LIN {X 0.007,Y -492.244,Z 296.515,A 0.000,B 0.000,C 90.000,E1 92.694} C_DIS
LIN {X -0.206,Y -481.791,Z 296.508,A 0.000,B 0.000,C 90.000,E1 91.489} C_DIS
LIN {X 0.068,Y -463.300,Z 296.496,A 0.000,B 0.000,C 90.000,E1 89.198} C_DIS
LIN {X 0.125,Y -448.239,Z 296.484,A 0.000,B 0.000,C 90.000,E1 87.135} C_DIS
LIN {X -0.046,Y -429.508,Z 296.468,A 0.000,B 0.000,C 90.000,E1 84.261} C_DIS
LIN {X 0.061,Y -414.133,Z 296.453,A 0.000,B 0.000,C 90.000,E1 81.546} C_DIS
LIN {X 0.059,Y -402.732,Z 296.441,A 0.000,B 0.000,C 90.000,E1 79.342} C_DIS
LIN {X 0.183,Y -394.078,Z 296.432,A 0.000,B 0.000,C 90.000,E1 77.645} C_DIS
LIN {X -0.138,Y -385.412,Z 296.422,A 0.000,B 0.000,C 90.000,E1 75.992} C_DIS
LIN {X -0.115,Y -373.962,Z 296.409,A 0.000,B 0.000,C 90.000,E1 73.685} C_DIS
LIN {X -0.134,Y -363.880,Z 296.398,A 0.000,B 0.000,C 90.000,E1 71.638} C_DIS
LIN {X 0.095,Y -353.920,Z 296.386,A 0.000,B 0.000,C 90.000,E1 69.518} C_DIS
LIN {X 0.073,Y -337.596,Z 296.366,A 0.000,B 0.000,C 90.000,E1 65.869} C_DIS
LIN {X 0.065,Y -324.350,Z 296.347,A 0.000,B 0.000,C 90.000,E1 62.436} C_DIS
LIN {X -0.104,Y -315.287,Z 296.333,A 0.000,B 0.000,C 90.000,E1 59.921} C_DIS
LIN {X -0.100,Y -307.615,Z 296.320,A 0.000,B 0.000,C 90.000,E1 57.661} C_DIS
LIN {X 0.046,Y -297.219,Z 296.302,A 0.000,B 0.000,C 90.000,E1 54.356} C_DIS
LIN {X 0.007,Y -289.192,Z 296.287,A 0.000,B 0.000,C 90.000,E1 51.698} C_DIS
LIN {X 0.042,Y -283.122,Z 296.276,A 0.000,B 0.000,C 90.000,E1 49.666} C_DIS
LIN {X -0.023,Y -275.077,Z 296.261,A 0.000,B 0.000,C 90.000,E1 46.944} C_DIS
LIN {X 0.007,Y -265.522,Z 296.241,A 0.000,B 0.000,C 90.000,E1 43.461} C_DIS
LIN {X -0.035,Y -259.977,Z 296.230,A 0.000,B 0.000,C 90.000,E1 41.353} C_DIS
LIN {X 0.039,Y -254.343,Z 296.218,A 0.000,B 0.000,C 90.000,E1 39.197} C_DIS
LIN {X 0.049,Y -248.620,Z 296.206,A 0.000,B 0.000,C 90.000,E1 37.030} C_DIS
LIN {X 0.150,Y -242.704,Z 296.194,A 0.000,B 0.000,C 90.000,E1 34.818} C_DIS
LIN {X 0.072,Y -234.757,Z 296.177,A 0.000,B 0.000,C 90.000,E1 31.878} C_DIS
LIN {X 0.072,Y -227.348,Z 296.160,A 0.000,B 0.000,C 90.000,E1 28.871} C_DIS
LIN {X -0.040,Y -220.568,Z 296.144,A 0.000,B 0.000,C 90.000,E1 25.848} C_DIS
LIN {X -0.103,Y -214.556,Z 296.126,A 0.000,B 0.000,C 90.000,E1 22.770} C_DIS
LIN {X -0.083,Y -209.396,Z 296.109,A 0.000,B 0.000,C 90.000,E1 19.631} C_DIS
LIN {X -0.069,Y -203.878,Z 296.087,A 0.000,B 0.000,C 90.000,E1 15.662} C_DIS
LIN {X -0.095,Y -199.386,Z 296.065,A 0.000,B 0.000,C 90.000,E1 11.658} C_DIS
LIN {X -0.019,Y -195.945,Z 296.042,A 0.000,B 0.000,C 90.000,E1 7.587} C_DIS
LIN {X -0.091,Y -192.735,Z 296.010,A 0.000,B 0.000,C 90.000,E1 1.892} C_DIS
LIN {X 0.075,Y -193.768,Z 295.924,A 0.000,B 0.000,C 90.000,E1 346.353} C_DIS
LIN {X 0.050,Y -197.101,Z 295.897,A 0.000,B 0.000,C 90.000,E1 341.456} C_DIS
LIN {X 0.012,Y -201.091,Z 295.875,A 0.000,B 0.000,C 90.000,E1 337.411} C_DIS
LIN {X 0.040,Y -206.121,Z 295.852,A 0.000,B 0.000,C 90.000,E1 333.384} C_DIS
LIN {X 0.043,Y -212.096,Z 295.830,A 0.000,B 0.000,C 90.000,E1 329.410} C_DIS
LIN {X -0.055,Y -217.536,Z 295.813,A 0.000,B 0.000,C 90.000,E1 326.294} C_DIS
LIN {X -0.005,Y -223.792,Z 295.795,A 0.000,B 0.000,C 90.000,E1 323.176} C_DIS
LIN {X -0.011,Y -230.919,Z 295.778,A 0.000,B 0.000,C 90.000,E1 320.114} C_DIS
LIN {X 0.094,Y -240.146,Z 295.760,A 0.000,B 0.000,C 90.000,E1 316.701} C_DIS
LIN {X 0.106,Y -250.567,Z 295.741,A 0.000,B 0.000,C 90.000,E1 313.380} C_DIS
LIN {X -0.081,Y -261.941,Z 295.723,A 0.000,B 0.000,C 90.000,E1 310.172} C_DIS
LIN {X -0.088,Y -274.440,Z 295.705,A 0.000,B 0.000,C 90.000,E1 306.996} C_DIS
LIN {X 0.098,Y -286.692,Z 295.690,A 0.000,B 0.000,C 90.000,E1 304.199} C_DIS
LIN {X -0.109,Y -300.388,Z 295.675,A 0.000,B 0.000,C 90.000,E1 301.544} C_DIS
LIN {X 0.043,Y -317.667,Z 295.659,A 0.000,B 0.000,C 90.000,E1 298.565} C_DIS
LIN {X -0.068,Y -338.547,Z 295.641,A 0.000,B 0.000,C 90.000,E1 295.412} C_DIS
LIN {X -0.100,Y -351.676,Z 295.631,A 0.000,B 0.000,C 90.000,E1 293.567} C_DIS
LIN {X -0.116,Y -367.035,Z 295.619,A 0.000,B 0.000,C 90.000,E1 291.461} C_DIS
LIN {X 0.211,Y -387.161,Z 295.604,A 0.000,B 0.000,C 90.000,E1 288.779} C_DIS
LIN {X 0.048,Y -400.967,Z 295.595,A 0.000,B 0.000,C 90.000,E1 287.094} C_DIS
LIN {X 0.126,Y -417.070,Z 295.584,A 0.000,B 0.000,C 90.000,E1 285.134} C_DIS
LIN {X -0.037,Y -426.115,Z 295.578,A 0.000,B 0.000,C 90.000,E1 284.064} C_DIS
LIN {X 0.045,Y -432.547,Z 295.574,A 0.000,B 0.000,C 90.000,E1 283.244} C_DIS
LIN {X -0.245,Y -438.494,Z 295.569,A 0.000,B 0.000,C 90.000,E1 282.479} C_DIS
LIN {X 0.172,Y -445.864,Z 295.563,A 0.000,B 0.000,C 90.000,E1 281.366} C_DIS
LIN {X -0.203,Y -452.680,Z 295.557,A 0.000,B 0.000,C 90.000,E1 280.366} C_DIS
LIN {X -0.143,Y -459.011,Z 295.552,A 0.000,B 0.000,C 90.000,E1 279.321} C_DIS
LIN {X -0.242,Y -466.365,Z 295.545,A 0.000,B 0.000,C 90.000,E1 278.049} C_DIS
LIN {X -0.237,Y -473.277,Z 295.537,A 0.000,B 0.000,C 90.000,E1 276.777} C_DIS
LIN {X 0.007,Y -478.221,Z 295.532,A 0.000,B 0.000,C 90.000,E1 275.739} C_DIS
LIN {X 0.151,Y -480.414,Z 295.529,A 0.000,B 0.000,C 90.000,E1 275.220} C_DIS
LIN {X -0.172,Y -482.241,Z 295.526,A 0.000,B 0.000,C 90.000,E1 274.759} C_DIS
LIN {X -0.046,Y -483.683,Z 295.524,A 0.000,B 0.000,C 90.000,E1 274.245} C_DIS
LIN {X 0.128,Y -484.744,Z 295.521,A 0.000,B 0.000,C 90.000,E1 273.726} C_DIS
LIN {X -0.207,Y -485.401,Z 295.518,A 0.000,B 0.000,C 90.000,E1 273.269} C_DIS
LIN {X -0.022,Y -485.681,Z 295.515,A 0.000,B 0.000,C 90.000,E1 272.751} C_DIS
LIN {X 0.143,Y -485.660,Z 295.513,A 0.000,B 0.000,C 90.000,E1 272.236} C_DIS
LIN {X 0.008,Y -484.956,Z 295.507,A 0.000,B 0.000,C 90.000,E1 271.260} C_DIS
LIN {X 0.174,Y -484.488,Z 295.504,A 0.000,B 0.000,C 90.000,E1 270.745} C_DIS
LIN {X -0.145,Y -483.841,Z 295.501,A 0.000,B 0.000,C 90.000,E1 270.286} C_DIS
LIN {X 0.017,Y -482.826,Z 295.499,A 0.000,B 0.000,C 90.000,E1 269.771} C_DIS
LIN {X 0.175,Y -481.325,Z 295.496,A 0.000,B 0.000,C 90.000,E1 269.255} C_DIS
LIN {X -0.155,Y -479.264,Z 295.493,A 0.000,B 0.000,C 90.000,E1 268.797} C_DIS
LIN {X -0.015,Y -476.458,Z 295.490,A 0.000,B 0.000,C 90.000,E1 268.282} C_DIS
LIN {X 0.121,Y -472.730,Z 295.488,A 0.000,B 0.000,C 90.000,E1 267.764} C_DIS
LIN {X -0.064,Y -470.502,Z 295.486,A 0.000,B 0.000,C 90.000,E1 267.535} C_DIS
LIN {X 0.094,Y -465.159,Z 295.484,A 0.000,B 0.000,C 90.000,E1 267.020} C_DIS
LIN {X -0.006,Y -462.035,Z 295.482,A 0.000,B 0.000,C 90.000,E1 266.788} C_DIS
LIN {X 0.135,Y -458.909,Z 295.481,A 0.000,B 0.000,C 90.000,E1 266.560} C_DIS
LIN {X -0.155,Y -452.026,Z 295.479,A 0.000,B 0.000,C 90.000,E1 266.216} C_DIS
LIN {X 0.191,Y -444.723,Z 295.477,A 0.000,B 0.000,C 90.000,E1 265.869} C_DIS
LIN {X 0.179,Y -436.512,Z 295.476,A 0.000,B 0.000,C 90.000,E1 265.641} C_DIS
LIN {X -0.133,Y -427.301,Z 295.475,A 0.000,B 0.000,C 90.000,E1 265.527} C_DIS
LIN {X 0.203,Y -418.825,Z 295.475,A 0.000,B 0.000,C 90.000,E1 265.412} C_DIS
LIN {X 0.062,Y -180.907,Z 295.475,A 0.000,B 0.000,C 90.000,E1 265.412} C_DIS
LIN {X -0.019,Y -180.696,Z 295.470,A 0.000,B 0.000,C 90.000,E1 264.546} C_DIS
LIN {X 0.059,Y -178.780,Z 295.442,A 0.000,B 0.000,C 90.000,E1 259.454} C_DIS
LIN {X -0.039,Y -175.826,Z 295.413,A 0.000,B 0.000,C 90.000,E1 254.393} C_DIS
LIN {X -0.038,Y -172.015,Z 295.385,A 0.000,B 0.000,C 90.000,E1 249.263} C_DIS
LIN {X -0.062,Y -171.436,Z 295.380,A 0.000,B 0.000,C 90.000,E1 248.411} C_DIS
LIN {X -0.007,Y -167.672,Z 295.356,A 0.000,B 0.000,C 90.000,E1 244.076} C_DIS
LIN {X -0.066,Y -166.346,Z 295.346,A 0.000,B 0.000,C 90.000,E1 242.359} C_DIS
LIN {X -0.074,Y -163.081,Z 295.327,A 0.000,B 0.000,C 90.000,E1 238.869} C_DIS
LIN {X -0.022,Y -161.023,Z 295.312,A 0.000,B 0.000,C 90.000,E1 236.215} C_DIS
LIN {X -0.039,Y -157.764,Z 295.293,A 0.000,B 0.000,C 90.000,E1 232.683} C_DIS
LIN {X 0.025,Y -155.802,Z 295.278,A 0.000,B 0.000,C 90.000,E1 229.989} C_DIS
LIN {X 0.079,Y -152.055,Z 295.253,A 0.000,B 0.000,C 90.000,E1 225.486} C_DIS
LIN {X -0.014,Y -150.304,Z 295.238,A 0.000,B 0.000,C 90.000,E1 222.813} C_DIS
LIN {X 0.022,Y -147.048,Z 295.213,A 0.000,B 0.000,C 90.000,E1 218.257} C_DIS
LIN {X 0.014,Y -145.627,Z 295.197,A 0.000,B 0.000,C 90.000,E1 215.518} C_DIS
LIN {X 0.012,Y -143.011,Z 295.172,A 0.000,B 0.000,C 90.000,E1 210.924} C_DIS
LIN {X -0.056,Y -141.637,Z 295.151,A 0.000,B 0.000,C 90.000,E1 207.257} C_DIS
LIN {X -0.006,Y -139.438,Z 295.115,A 0.000,B 0.000,C 90.000,E1 200.737} C_DIS
LIN {X 0.049,Y -139.170,Z 295.105,A 0.000,B 0.000,C 90.000,E1 198.852} C_DIS
LIN {X -0.055,Y -138.317,Z 295.053,A 0.000,B 0.000,C 90.000,E1 189.557} C_DIS
LIN {X -0.046,Y -139.473,Z 295.006,A 0.000,B 0.000,C 90.000,E1 181.146} C_DIS
LIN {X 0.034,Y -141.049,Z 294.975,A 0.000,B 0.000,C 90.000,E1 175.527} C_DIS
LIN {X -0.012,Y -142.420,Z 294.960,A 0.000,B 0.000,C 90.000,E1 172.761} C_DIS
LIN {X 0.050,Y -144.656,Z 294.934,A 0.000,B 0.000,C 90.000,E1 168.117} C_DIS
LIN {X -0.032,Y -147.852,Z 294.909,A 0.000,B 0.000,C 90.000,E1 163.559} C_DIS
LIN {X 0.053,Y -150.553,Z 294.888,A 0.000,B 0.000,C 90.000,E1 159.880} C_DIS
LIN {X -0.070,Y -154.020,Z 294.868,A 0.000,B 0.000,C 90.000,E1 156.305} C_DIS
LIN {X -0.011,Y -157.436,Z 294.848,A 0.000,B 0.000,C 90.000,E1 152.692} C_DIS
LIN {X 0.010,Y -161.650,Z 294.828,A 0.000,B 0.000,C 90.000,E1 149.125} C_DIS
LIN {X 0.027,Y -165.845,Z 294.809,A 0.000,B 0.000,C 90.000,E1 145.595} C_DIS
LIN {X 0.020,Y -170.819,Z 294.790,A 0.000,B 0.000,C 90.000,E1 142.110} C_DIS
LIN {X -0.064,Y -175.689,Z 294.770,A 0.000,B 0.000,C 90.000,E1 138.690} C_DIS
LIN {X 0.059,Y -181.301,Z 294.751,A 0.000,B 0.000,C 90.000,E1 135.243} C_DIS
LIN {X -0.069,Y -186.783,Z 294.733,A 0.000,B 0.000,C 90.000,E1 131.919} C_DIS
LIN {X 0.002,Y -191.375,Z 294.719,A 0.000,B 0.000,C 90.000,E1 129.402} C_DIS
LIN {X 0.085,Y -197.217,Z 294.701,A 0.000,B 0.000,C 90.000,E1 126.091} C_DIS
LIN {X 0.009,Y -200.494,Z 294.692,A 0.000,B 0.000,C 90.000,E1 124.485} C_DIS
LIN {X 0.109,Y -202.532,Z 294.685,A 0.000,B 0.000,C 90.000,E1 123.293} C_DIS
LIN {X 0.119,Y -304.407,Z 294.685,A 0.000,B 0.000,C 90.000,E1 123.293} C_DIS
LIN {X -0.015,Y -305.950,Z 294.685,A 0.000,B 0.000,C 90.000,E1 123.293} C_DIS
LIN {X -0.030,Y -310.535,Z 294.684,A 0.000,B 0.000,C 90.000,E1 123.086} C_DIS
LIN {X -0.046,Y -313.045,Z 294.683,A 0.000,B 0.000,C 90.000,E1 122.880} C_DIS
LIN {X -0.182,Y -316.856,Z 294.680,A 0.000,B 0.000,C 90.000,E1 122.418} C_DIS
LIN {X -0.123,Y -318.617,Z 294.678,A 0.000,B 0.000,C 90.000,E1 122.084} C_DIS
LIN {X 0.016,Y -321.157,Z 294.675,A 0.000,B 0.000,C 90.000,E1 121.416} C_DIS
LIN {X 0.002,Y -332.328,Z 294.659,A 0.000,B 0.000,C 90.000,E1 118.565} C_DIS
LIN {X -0.018,Y -344.918,Z 294.643,A 0.000,B 0.000,C 90.000,E1 115.771} C_DIS
LIN {X -0.013,Y -357.397,Z 294.630,A 0.000,B 0.000,C 90.000,E1 113.334} C_DIS
LIN {X 0.185,Y -371.181,Z 294.616,A 0.000,B 0.000,C 90.000,E1 110.918} C_DIS
LIN {X 0.115,Y -386.373,Z 294.603,A 0.000,B 0.000,C 90.000,E1 108.598} C_DIS
LIN {X 0.171,Y -403.084,Z 294.591,A 0.000,B 0.000,C 90.000,E1 106.315} C_DIS
LIN {X 0.025,Y -421.438,Z 294.578,A 0.000,B 0.000,C 90.000,E1 104.120} C_DIS
LIN {X -0.070,Y -441.277,Z 294.567,A 0.000,B 0.000,C 90.000,E1 102.007} C_DIS
LIN {X 0.214,Y -461.762,Z 294.556,A 0.000,B 0.000,C 90.000,E1 100.018} C_DIS
LIN {X -0.085,Y -485.422,Z 294.545,A 0.000,B 0.000,C 90.000,E1 98.049} C_DIS
LIN {X 0.021,Y -498.737,Z 294.539,A 0.000,B 0.000,C 90.000,E1 97.004} C_DIS
LIN {X 0.249,Y -500.822,Z 294.538,A 0.000,B 0.000,C 90.000,E1 96.777} C_DIS
LIN {X 0.176,Y -502.677,Z 294.536,A 0.000,B 0.000,C 90.000,E1 96.549} C_DIS
LIN {X 0.158,Y -504.077,Z 294.535,A 0.000,B 0.000,C 90.000,E1 96.315} C_DIS
LIN {X -0.042,Y -505.916,Z 294.533,A 0.000,B 0.000,C 90.000,E1 95.853} C_DIS
LIN {X 0.269,Y -506.626,Z 294.530,A 0.000,B 0.000,C 90.000,E1 95.334} C_DIS
LIN {X 0.040,Y -506.327,Z 294.527,A 0.000,B 0.000,C 90.000,E1 94.878} C_DIS
LIN {X -0.139,Y -504.971,Z 294.524,A 0.000,B 0.000,C 90.000,E1 94.416} C_DIS
LIN {X -0.249,Y -503.823,Z 294.523,A 0.000,B 0.000,C 90.000,E1 94.188} C_DIS
LIN {X 0.178,Y -502.279,Z 294.522,A 0.000,B 0.000,C 90.000,E1 93.898} C_DIS
LIN {X 0.226,Y -494.728,Z 294.516,A 0.000,B 0.000,C 90.000,E1 92.922} C_DIS
LIN {X 0.036,Y -484.399,Z 294.510,A 0.000,B 0.000,C 90.000,E1 91.718} C_DIS
LIN {X 0.167,Y -463.746,Z 294.496,A 0.000,B 0.000,C 90.000,E1 89.198} C_DIS
LIN {X -0.216,Y -448.648,Z 294.484,A 0.000,B 0.000,C 90.000,E1 87.192} C_DIS
LIN {X -0.227,Y -428.267,Z 294.467,A 0.000,B 0.000,C 90.000,E1 84.033} C_DIS
LIN {X -0.095,Y -413.022,Z 294.452,A 0.000,B 0.000,C 90.000,E1 81.310} C_DIS
LIN {X -0.114,Y -401.654,Z 294.439,A 0.000,B 0.000,C 90.000,E1 79.106} C_DIS
LIN {X 0.063,Y -391.543,Z 294.428,A 0.000,B 0.000,C 90.000,E1 77.117} C_DIS
LIN {X -0.139,Y -380.032,Z 294.416,A 0.000,B 0.000,C 90.000,E1 74.866} C_DIS
LIN {X -0.132,Y -370.007,Z 294.405,A 0.000,B 0.000,C 90.000,E1 72.834} C_DIS
LIN {X 0.184,Y -358.557,Z 294.391,A 0.000,B 0.000,C 90.000,E1 70.423} C_DIS
LIN {X 0.017,Y -345.956,Z 294.376,A 0.000,B 0.000,C 90.000,E1 67.741} C_DIS
LIN {X 0.035,Y -334.235,Z 294.361,A 0.000,B 0.000,C 90.000,E1 64.973} C_DIS
LIN {X 0.078,Y -321.330,Z 294.342,A 0.000,B 0.000,C 90.000,E1 61.513} C_DIS
LIN {X -0.037,Y -310.212,Z 294.324,A 0.000,B 0.000,C 90.000,E1 58.329} C_DIS
LIN {X 0.030,Y -299.658,Z 294.306,A 0.000,B 0.000,C 90.000,E1 55.055} C_DIS
LIN {X 0.054,Y -291.573,Z 294.291,A 0.000,B 0.000,C 90.000,E1 52.396} C_DIS
LIN {X 0.177,Y -285.517,Z 294.280,A 0.000,B 0.000,C 90.000,E1 50.356} C_DIS
LIN {X -0.039,Y -277.399,Z 294.265,A 0.000,B 0.000,C 90.000,E1 47.676} C_DIS
LIN {X 0.075,Y -267.698,Z 294.246,A 0.000,B 0.000,C 90.000,E1 44.190} C_DIS
LIN {X 0.077,Y -262.142,Z 294.234,A 0.000,B 0.000,C 90.000,E1 42.081} C_DIS
LIN {X -0.001,Y -256.552,Z 294.222,A 0.000,B 0.000,C 90.000,E1 39.967} C_DIS
LIN {X 0.013,Y -250.884,Z 294.210,A 0.000,B 0.000,C 90.000,E1 37.810} C_DIS
LIN {X -0.043,Y -245.007,Z 294.198,A 0.000,B 0.000,C 90.000,E1 35.644} C_DIS
LIN {X 0.043,Y -239.047,Z 294.186,A 0.000,B 0.000,C 90.000,E1 33.420} C_DIS
LIN {X -0.050,Y -231.258,Z 294.169,A 0.000,B 0.000,C 90.000,E1 30.463} C_DIS
LIN {X -0.035,Y -222.505,Z 294.148,A 0.000,B 0.000,C 90.000,E1 26.668} C_DIS
LIN {X -0.088,Y -214.899,Z 294.127,A 0.000,B 0.000,C 90.000,E1 22.823} C_DIS
LIN {X -0.063,Y -209.719,Z 294.109,A 0.000,B 0.000,C 90.000,E1 19.685} C_DIS
LIN {X -0.045,Y -204.183,Z 294.087,A 0.000,B 0.000,C 90.000,E1 15.717} C_DIS
LIN {X -0.065,Y -199.679,Z 294.065,A 0.000,B 0.000,C 90.000,E1 11.715} C_DIS
LIN {X 0.017,Y -196.219,Z 294.042,A 0.000,B 0.000,C 90.000,E1 7.644} C_DIS
LIN {X -0.046,Y -192.989,Z 294.011,A 0.000,B 0.000,C 90.000,E1 1.949} C_DIS
LIN {X -0.093,Y -193.946,Z 293.924,A 0.000,B 0.000,C 90.000,E1 346.408} C_DIS
LIN {X 0.076,Y -197.236,Z 293.897,A 0.000,B 0.000,C 90.000,E1 341.456} C_DIS
LIN {X 0.043,Y -201.224,Z 293.875,A 0.000,B 0.000,C 90.000,E1 337.411} C_DIS
LIN {X 0.077,Y -206.253,Z 293.852,A 0.000,B 0.000,C 90.000,E1 333.384} C_DIS
LIN {X 0.085,Y -212.202,Z 293.830,A 0.000,B 0.000,C 90.000,E1 329.410} C_DIS
LIN {X -0.010,Y -217.665,Z 293.813,A 0.000,B 0.000,C 90.000,E1 326.294} C_DIS
LIN {X -0.089,Y -223.938,Z 293.795,A 0.000,B 0.000,C 90.000,E1 323.210} C_DIS
LIN {X 0.045,Y -231.110,Z 293.778,A 0.000,B 0.000,C 90.000,E1 320.114} C_DIS
LIN {X -0.017,Y -240.364,Z 293.760,A 0.000,B 0.000,C 90.000,E1 316.743} C_DIS
LIN {X 0.007,Y -250.757,Z 293.741,A 0.000,B 0.000,C 90.000,E1 313.419} C_DIS
LIN {X 0.000,Y -262.119,Z 293.723,A 0.000,B 0.000,C 90.000,E1 310.172} C_DIS
LIN {X 0.003,Y -274.632,Z 293.706,A 0.000,B 0.000,C 90.000,E1 306.996} C_DIS
LIN {X -0.039,Y -286.899,Z 293.690,A 0.000,B 0.000,C 90.000,E1 304.246} C_DIS
LIN {X 0.000,Y -300.617,Z 293.675,A 0.000,B 0.000,C 90.000,E1 301.544} C_DIS
LIN {X -0.113,Y -317.889,Z 293.659,A 0.000,B 0.000,C 90.000,E1 298.615} C_DIS
LIN {X 0.070,Y -338.772,Z 293.641,A 0.000,B 0.000,C 90.000,E1 295.412} C_DIS
LIN {X 0.047,Y -351.870,Z 293.631,A 0.000,B 0.000,C 90.000,E1 293.567} C_DIS
LIN {X 0.042,Y -367.202,Z 293.619,A 0.000,B 0.000,C 90.000,E1 291.461} C_DIS
LIN {X 0.027,Y -389.558,Z 293.603,A 0.000,B 0.000,C 90.000,E1 288.544} C_DIS
LIN {X -0.096,Y -403.296,Z 293.594,A 0.000,B 0.000,C 90.000,E1 286.858} C_DIS
LIN {X 0.036,Y -419.280,Z 293.583,A 0.000,B 0.000,C 90.000,E1 284.898} C_DIS
LIN {X -0.102,Y -428.214,Z 293.577,A 0.000,B 0.000,C 90.000,E1 283.828} C_DIS
LIN {X -0.009,Y -434.477,Z 293.572,A 0.000,B 0.000,C 90.000,E1 283.008} C_DIS
LIN {X -0.072,Y -442.119,Z 293.566,A 0.000,B 0.000,C 90.000,E1 281.951} C_DIS
LIN {X -0.048,Y -449.158,Z 293.560,A 0.000,B 0.000,C 90.000,E1 280.894} C_DIS
LIN {X -0.026,Y -455.719,Z 293.555,A 0.000,B 0.000,C 90.000,E1 279.849} C_DIS
LIN {X -0.097,Y -463.283,Z 293.548,A 0.000,B 0.000,C 90.000,E1 278.568} C_DIS
LIN {X 0.116,Y -471.739,Z 293.539,A 0.000,B 0.000,C 90.000,E1 277.011} C_DIS
LIN {X -0.125,Y -476.861,Z 293.533,A 0.000,B 0.000,C 90.000,E1 276.030} C_DIS
LIN {X -0.130,Y -480.211,Z 293.529,A 0.000,B 0.000,C 90.000,E1 275.277} C_DIS
LIN {X 0.024,Y -482.082,Z 293.526,A 0.000,B 0.000,C 90.000,E1 274.759} C_DIS
LIN {X 0.148,Y -483.513,Z 293.524,A 0.000,B 0.000,C 90.000,E1 274.245} C_DIS
LIN {X -0.162,Y -484.596,Z 293.521,A 0.000,B 0.000,C 90.000,E1 273.784} C_DIS
LIN {X -0.012,Y -485.230,Z 293.518,A 0.000,B 0.000,C 90.000,E1 273.269} C_DIS
LIN {X 0.171,Y -485.559,Z 293.515,A 0.000,B 0.000,C 90.000,E1 272.751} C_DIS
LIN {X -0.151,Y -485.544,Z 293.513,A 0.000,B 0.000,C 90.000,E1 272.293} C_DIS
LIN {X 0.198,Y -484.896,Z 293.507,A 0.000,B 0.000,C 90.000,E1 271.260} C_DIS
LIN {X 0.044,Y -483.782,Z 293.502,A 0.000,B 0.000,C 90.000,E1 270.286} C_DIS
LIN {X 0.205,Y -482.822,Z 293.499,A 0.000,B 0.000,C 90.000,E1 269.771} C_DIS
LIN {X -0.119,Y -481.361,Z 293.496,A 0.000,B 0.000,C 90.000,E1 269.312} C_DIS
LIN {X 0.032,Y -479.303,Z 293.493,A 0.000,B 0.000,C 90.000,E1 268.797} C_DIS
LIN {X 0.172,Y -476.535,Z 293.491,A 0.000,B 0.000,C 90.000,E1 268.282} C_DIS
LIN {X 0.009,Y -474.850,Z 293.489,A 0.000,B 0.000,C 90.000,E1 268.051} C_DIS
LIN {X 0.121,Y -470.648,Z 293.486,A 0.000,B 0.000,C 90.000,E1 267.535} C_DIS
LIN {X -0.065,Y -468.184,Z 293.485,A 0.000,B 0.000,C 90.000,E1 267.306} C_DIS
LIN {X -0.240,Y -465.387,Z 293.484,A 0.000,B 0.000,C 90.000,E1 267.078} C_DIS
LIN {X 0.073,Y -462.253,Z 293.482,A 0.000,B 0.000,C 90.000,E1 266.788} C_DIS
LIN {X 0.186,Y -459.176,Z 293.481,A 0.000,B 0.000,C 90.000,E1 266.560} C_DIS
LIN {X -0.157,Y -455.611,Z 293.480,A 0.000,B 0.000,C 90.000,E1 266.388} C_DIS
LIN {X -0.188,Y -448.440,Z 293.478,A 0.000,B 0.000,C 90.000,E1 266.045} C_DIS
LIN {X 0.114,Y -444.902,Z 293.477,A 0.000,B 0.000,C 90.000,E1 265.869} C_DIS
LIN {X 0.077,Y -436.623,Z 293.476,A 0.000,B 0.000,C 90.000,E1 265.641} C_DIS
LIN {X 0.181,Y -427.335,Z 293.475,A 0.000,B 0.000,C 90.000,E1 265.469} C_DIS
LIN {X 0.083,Y -417.648,Z 293.475,A 0.000,B 0.000,C 90.000,E1 265.412} C_DIS
LIN {X 0.008,Y -180.906,Z 293.475,A 0.000,B 0.000,C 90.000,E1 265.412} C_DIS
LIN {X 0.089,Y -180.684,Z 293.470,A 0.000,B 0.000,C 90.000,E1 264.489} C_DIS
LIN {X -0.013,Y -178.767,Z 293.441,A 0.000,B 0.000,C 90.000,E1 259.454} C_DIS
LIN {X 0.059,Y -175.814,Z 293.413,A 0.000,B 0.000,C 90.000,E1 254.338} C_DIS
LIN {X 0.052,Y -172.001,Z 293.385,A 0.000,B 0.000,C 90.000,E1 249.209} C_DIS
LIN {X 0.027,Y -171.416,Z 293.380,A 0.000,B 0.000,C 90.000,E1 248.358} C_DIS
LIN {X 0.074,Y -167.654,Z 293.356,A 0.000,B 0.000,C 90.000,E1 244.024} C_DIS
LIN {X 0.089,Y -166.321,Z 293.346,A 0.000,B 0.000,C 90.000,E1 242.281} C_DIS
LIN {X -0.002,Y -163.061,Z 293.327,A 0.000,B 0.000,C 90.000,E1 238.820} C_DIS
LIN {X 0.043,Y -160.998,Z 293.312,A 0.000,B 0.000,C 90.000,E1 236.167} C_DIS
LIN {X 0.020,Y -157.744,Z 293.292,A 0.000,B 0.000,C 90.000,E1 232.637} C_DIS
LIN {X -0.041,Y -155.783,Z 293.278,A 0.000,B 0.000,C 90.000,E1 229.989} C_DIS
LIN {X 0.014,Y -152.036,Z 293.253,A 0.000,B 0.000,C 90.000,E1 225.486} C_DIS
LIN {X 0.032,Y -150.285,Z 293.238,A 0.000,B 0.000,C 90.000,E1 222.771} C_DIS
LIN {X -0.043,Y -147.035,Z 293.212,A 0.000,B 0.000,C 90.000,E1 218.257} C_DIS
LIN {X -0.050,Y -145.615,Z 293.197,A 0.000,B 0.000,C 90.000,E1 215.518} C_DIS
LIN {X -0.050,Y -142.999,Z 293.172,A 0.000,B 0.000,C 90.000,E1 210.924} C_DIS
LIN {X 0.007,Y -141.626,Z 293.151,A 0.000,B 0.000,C 90.000,E1 207.206} C_DIS
LIN {X -0.068,Y -139.433,Z 293.115,A 0.000,B 0.000,C 90.000,E1 200.737} C_DIS
LIN {X -0.014,Y -139.165,Z 293.105,A 0.000,B 0.000,C 90.000,E1 198.852} C_DIS
LIN {X 0.019,Y -138.316,Z 293.053,A 0.000,B 0.000,C 90.000,E1 189.500} C_DIS
LIN {X 0.031,Y -139.477,Z 293.006,A 0.000,B 0.000,C 90.000,E1 181.088} C_DIS
LIN {X -0.028,Y -141.060,Z 292.975,A 0.000,B 0.000,C 90.000,E1 175.527} C_DIS
LIN {X 0.067,Y -142.433,Z 292.960,A 0.000,B 0.000,C 90.000,E1 172.704} C_DIS
LIN {X -0.013,Y -144.671,Z 292.934,A 0.000,B 0.000,C 90.000,E1 168.117} C_DIS
LIN {X -0.030,Y -147.256,Z 292.914,A 0.000,B 0.000,C 90.000,E1 164.448} C_DIS
LIN {X -0.013,Y -150.574,Z 292.888,A 0.000,B 0.000,C 90.000,E1 159.880} C_DIS
LIN {X 0.066,Y -154.044,Z 292.868,A 0.000,B 0.000,C 90.000,E1 156.230} C_DIS
LIN {X -0.007,Y -157.462,Z 292.848,A 0.000,B 0.000,C 90.000,E1 152.666} C_DIS
LIN {X -0.059,Y -161.682,Z 292.828,A 0.000,B 0.000,C 90.000,E1 149.125} C_DIS
LIN {X -0.042,Y -165.877,Z 292.809,A 0.000,B 0.000,C 90.000,E1 145.595} C_DIS
LIN {X -0.051,Y -170.855,Z 292.789,A 0.000,B 0.000,C 90.000,E1 142.110} C_DIS
LIN {X -0.004,Y -175.725,Z 292.770,A 0.000,B 0.000,C 90.000,E1 138.647} C_DIS
LIN {X -0.014,Y -181.336,Z 292.751,A 0.000,B 0.000,C 90.000,E1 135.243} C_DIS
LIN {X -0.019,Y -186.823,Z 292.733,A 0.000,B 0.000,C 90.000,E1 131.881} C_DIS
LIN {X 0.075,Y -191.412,Z 292.719,A 0.000,B 0.000,C 90.000,E1 129.358} C_DIS
LIN {X 0.008,Y -197.260,Z 292.701,A 0.000,B 0.000,C 90.000,E1 126.091} C_DIS
LIN {X -0.068,Y -200.538,Z 292.691,A 0.000,B 0.000,C 90.000,E1 124.485} C_DIS
LIN {X -0.030,Y -202.602,Z 292.685,A 0.000,B 0.000,C 90.000,E1 123.293} C_DIS
LIN {X -0.089,Y -304.500,Z 292.685,A 0.000,B 0.000,C 90.000,E1 123.293} C_DIS
LIN {X 0.110,Y -310.380,Z 292.684,A 0.000,B 0.000,C 90.000,E1 123.038} C_DIS
LIN {X 0.096,Y -312.969,Z 292.682,A 0.000,B 0.000,C 90.000,E1 122.832} C_DIS
LIN {X 0.202,Y -316.775,Z 292.680,A 0.000,B 0.000,C 90.000,E1 122.339} C_DIS
LIN {X -0.008,Y -318.585,Z 292.678,A 0.000,B 0.000,C 90.000,E1 122.054} C_DIS
LIN {X -0.038,Y -321.171,Z 292.674,A 0.000,B 0.000,C 90.000,E1 121.416} C_DIS
LIN {X -0.053,Y -332.347,Z 292.659,A 0.000,B 0.000,C 90.000,E1 118.565} C_DIS
LIN {X -0.076,Y -344.941,Z 292.643,A 0.000,B 0.000,C 90.000,E1 115.771} C_DIS
LIN {X -0.072,Y -357.425,Z 292.630,A 0.000,B 0.000,C 90.000,E1 113.334} C_DIS
LIN {X 0.124,Y -371.214,Z 292.616,A 0.000,B 0.000,C 90.000,E1 110.918} C_DIS
LIN {X 0.052,Y -386.411,Z 292.603,A 0.000,B 0.000,C 90.000,E1 108.598} C_DIS
LIN {X 0.107,Y -403.128,Z 292.591,A 0.000,B 0.000,C 90.000,E1 106.315} C_DIS
LIN {X -0.041,Y -421.490,Z 292.578,A 0.000,B 0.000,C 90.000,E1 104.120} C_DIS
LIN {X -0.135,Y -441.333,Z 292.567,A 0.000,B 0.000,C 90.000,E1 102.007} C_DIS
LIN {X 0.151,Y -461.819,Z 292.556,A 0.000,B 0.000,C 90.000,E1 100.018} C_DIS
LIN {X -0.147,Y -485.482,Z 292.545,A 0.000,B 0.000,C 90.000,E1 98.049} C_DIS
LIN {X -0.041,Y -498.817,Z 292.539,A 0.000,B 0.000,C 90.000,E1 97.004} C_DIS
LIN {X 0.188,Y -500.942,Z 292.538,A 0.000,B 0.000,C 90.000,E1 96.777} C_DIS
LIN {X 0.138,Y -502.807,Z 292.536,A 0.000,B 0.000,C 90.000,E1 96.549} C_DIS
LIN {X 0.144,Y -504.220,Z 292.535,A 0.000,B 0.000,C 90.000,E1 96.315} C_DIS
LIN {X -0.055,Y -506.099,Z 292.532,A 0.000,B 0.000,C 90.000,E1 95.853} C_DIS
LIN {X 0.256,Y -506.844,Z 292.530,A 0.000,B 0.000,C 90.000,E1 95.334} C_DIS
LIN {X 0.028,Y -506.581,Z 292.527,A 0.000,B 0.000,C 90.000,E1 94.878} C_DIS
LIN {X -0.150,Y -505.265,Z 292.524,A 0.000,B 0.000,C 90.000,E1 94.416} C_DIS
LIN {X -0.259,Y -504.142,Z 292.523,A 0.000,B 0.000,C 90.000,E1 94.188} C_DIS
LIN {X 0.169,Y -502.628,Z 292.522,A 0.000,B 0.000,C 90.000,E1 93.898} C_DIS
LIN {X -0.180,Y -497.073,Z 292.518,A 0.000,B 0.000,C 90.000,E1 93.212} C_DIS
LIN {X -0.180,Y -489.032,Z 292.512,A 0.000,B 0.000,C 90.000,E1 92.236} C_DIS
LIN {X -0.086,Y -466.089,Z 292.497,A 0.000,B 0.000,C 90.000,E1 89.484} C_DIS
LIN {X -0.181,Y -452.605,Z 292.487,A 0.000,B 0.000,C 90.000,E1 87.707} C_DIS
LIN {X 0.197,Y -433.472,Z 292.471,A 0.000,B 0.000,C 90.000,E1 84.780} C_DIS
LIN {X -0.063,Y -417.699,Z 292.456,A 0.000,B 0.000,C 90.000,E1 82.129} C_DIS
LIN {X 0.120,Y -404.773,Z 292.443,A 0.000,B 0.000,C 90.000,E1 79.634} C_DIS
LIN {X -0.109,Y -396.170,Z 292.433,A 0.000,B 0.000,C 90.000,E1 77.993} C_DIS
LIN {X 0.043,Y -386.081,Z 292.422,A 0.000,B 0.000,C 90.000,E1 75.992} C_DIS
LIN {X 0.077,Y -374.626,Z 292.409,A 0.000,B 0.000,C 90.000,E1 73.685} C_DIS
LIN {X 0.067,Y -364.566,Z 292.398,A 0.000,B 0.000,C 90.000,E1 71.638} C_DIS
LIN {X 0.022,Y -353.232,Z 292.385,A 0.000,B 0.000,C 90.000,E1 69.263} C_DIS
LIN {X -0.012,Y -337.089,Z 292.365,A 0.000,B 0.000,C 90.000,E1 65.613} C_DIS
LIN {X 0.123,Y -323.953,Z 292.345,A 0.000,B 0.000,C 90.000,E1 62.153} C_DIS
LIN {X 0.067,Y -314.936,Z 292.331,A 0.000,B 0.000,C 90.000,E1 59.616} C_DIS
LIN {X 0.010,Y -306.224,Z 292.317,A 0.000,B 0.000,C 90.000,E1 57.041} C_DIS
LIN {X 0.095,Y -297.963,Z 292.302,A 0.000,B 0.000,C 90.000,E1 54.402} C_DIS
LIN {X -0.017,Y -291.910,Z 292.291,A 0.000,B 0.000,C 90.000,E1 52.431} C_DIS
LIN {X -0.115,Y -285.834,Z 292.280,A 0.000,B 0.000,C 90.000,E1 50.436} C_DIS
LIN {X -0.111,Y -277.690,Z 292.265,A 0.000,B 0.000,C 90.000,E1 47.715} C_DIS
LIN {X 0.003,Y -267.964,Z 292.246,A 0.000,B 0.000,C 90.000,E1 44.231} C_DIS
LIN {X -0.077,Y -260.560,Z 292.230,A 0.000,B 0.000,C 90.000,E1 41.434} C_DIS
LIN {X 0.009,Y -254.941,Z 292.218,A 0.000,B 0.000,C 90.000,E1 39.277} C_DIS
LIN {X 0.035,Y -249.256,Z 292.206,A 0.000,B 0.000,C 90.000,E1 37.111} C_DIS
LIN {X -0.051,Y -243.321,Z 292.194,A 0.000,B 0.000,C 90.000,E1 34.945} C_DIS
LIN {X -0.110,Y -235.368,Z 292.178,A 0.000,B 0.000,C 90.000,E1 32.005} C_DIS
LIN {X 0.108,Y -227.950,Z 292.161,A 0.000,B 0.000,C 90.000,E1 28.949} C_DIS
LIN {X 0.015,Y -221.205,Z 292.144,A 0.000,B 0.000,C 90.000,E1 25.924} C_DIS
LIN {X 0.055,Y -215.207,Z 292.127,A 0.000,B 0.000,C 90.000,E1 22.823} C_DIS
LIN {X 0.013,Y -210.013,Z 292.109,A 0.000,B 0.000,C 90.000,E1 19.704} C_DIS
LIN {X 0.051,Y -204.461,Z 292.087,A 0.000,B 0.000,C 90.000,E1 15.733} C_DIS
LIN {X 0.091,Y -199.945,Z 292.065,A 0.000,B 0.000,C 90.000,E1 11.715} C_DIS
LIN {X -0.025,Y -195.882,Z 292.038,A 0.000,B 0.000,C 90.000,E1 6.891} C_DIS
LIN {X 0.070,Y -192.920,Z 292.006,A 0.000,B 0.000,C 90.000,E1 1.146} C_DIS
LIN {X -0.074,Y -194.121,Z 291.924,A 0.000,B 0.000,C 90.000,E1 346.408} C_DIS
LIN {X 0.103,Y -197.383,Z 291.897,A 0.000,B 0.000,C 90.000,E1 341.456} C_DIS
LIN {X 0.075,Y -201.360,Z 291.875,A 0.000,B 0.000,C 90.000,E1 337.411} C_DIS
LIN {X 0.114,Y -206.386,Z 291.852,A 0.000,B 0.000,C 90.000,E1 333.384} C_DIS
LIN {X -0.056,Y -212.320,Z 291.830,A 0.000,B 0.000,C 90.000,E1 329.459} C_DIS
LIN {X 0.036,Y -217.796,Z 291.813,A 0.000,B 0.000,C 90.000,E1 326.294} C_DIS
LIN {X -0.038,Y -224.089,Z 291.796,A 0.000,B 0.000,C 90.000,E1 323.210} C_DIS
LIN {X -0.047,Y -231.302,Z 291.779,A 0.000,B 0.000,C 90.000,E1 320.150} C_DIS
LIN {X 0.047,Y -240.580,Z 291.760,A 0.000,B 0.000,C 90.000,E1 316.743} C_DIS
LIN {X -0.102,Y -250.951,Z 291.741,A 0.000,B 0.000,C 90.000,E1 313.461} C_DIS
LIN {X 0.083,Y -262.304,Z 291.723,A 0.000,B 0.000,C 90.000,E1 310.172} C_DIS
LIN {X -0.071,Y -274.816,Z 291.706,A 0.000,B 0.000,C 90.000,E1 307.030} C_DIS
LIN {X 0.061,Y -287.103,Z 291.690,A 0.000,B 0.000,C 90.000,E1 304.246} C_DIS
LIN {X 0.107,Y -299.024,Z 291.677,A 0.000,B 0.000,C 90.000,E1 301.878} C_DIS
LIN {X 0.011,Y -318.113,Z 291.659,A 0.000,B 0.000,C 90.000,E1 298.615} C_DIS
LIN {X -0.075,Y -336.840,Z 291.643,A 0.000,B 0.000,C 90.000,E1 295.771} C_DIS
LIN {X 0.056,Y -352.032,Z 291.631,A 0.000,B 0.000,C 90.000,E1 293.590} C_DIS
LIN {X 0.067,Y -367.354,Z 291.619,A 0.000,B 0.000,C 90.000,E1 291.482} C_DIS
LIN {X 0.062,Y -387.323,Z 291.605,A 0.000,B 0.000,C 90.000,E1 288.852} C_DIS
LIN {X 0.021,Y -401.056,Z 291.595,A 0.000,B 0.000,C 90.000,E1 287.149} C_DIS
LIN {X 0.096,Y -416.951,Z 291.584,A 0.000,B 0.000,C 90.000,E1 285.190} C_DIS
LIN {X 0.089,Y -428.112,Z 291.577,A 0.000,B 0.000,C 90.000,E1 283.828} C_DIS
LIN {X 0.184,Y -434.367,Z 291.572,A 0.000,B 0.000,C 90.000,E1 283.008} C_DIS
LIN {X 0.123,Y -441.967,Z 291.566,A 0.000,B 0.000,C 90.000,E1 281.951} C_DIS
LIN {X 0.148,Y -448.969,Z 291.561,A 0.000,B 0.000,C 90.000,E1 280.894} C_DIS
LIN {X 0.170,Y -455.524,Z 291.555,A 0.000,B 0.000,C 90.000,E1 279.849} C_DIS
LIN {X 0.100,Y -463.066,Z 291.548,A 0.000,B 0.000,C 90.000,E1 278.568} C_DIS
LIN {X 0.060,Y -470.156,Z 291.541,A 0.000,B 0.000,C 90.000,E1 277.296} C_DIS
LIN {X -0.202,Y -475.407,Z 291.535,A 0.000,B 0.000,C 90.000,E1 276.315} C_DIS
LIN {X 0.066,Y -480.003,Z 291.529,A 0.000,B 0.000,C 90.000,E1 275.277} C_DIS
LIN {X 0.220,Y -481.879,Z 291.527,A 0.000,B 0.000,C 90.000,E1 274.759} C_DIS
LIN {X -0.138,Y -483.339,Z 291.524,A 0.000,B 0.000,C 90.000,E1 274.302} C_DIS
LIN {X 0.033,Y -484.424,Z 291.521,A 0.000,B 0.000,C 90.000,E1 273.784} C_DIS
LIN {X 0.181,Y -485.086,Z 291.518,A 0.000,B 0.000,C 90.000,E1 273.269} C_DIS
LIN {X -0.121,Y -485.437,Z 291.516,A 0.000,B 0.000,C 90.000,E1 272.808} C_DIS
LIN {X 0.041,Y -485.448,Z 291.513,A 0.000,B 0.000,C 90.000,E1 272.293} C_DIS
LIN {X -0.096,Y -484.821,Z 291.507,A 0.000,B 0.000,C 90.000,E1 271.318} C_DIS
LIN {X 0.069,Y -484.387,Z 291.505,A 0.000,B 0.000,C 90.000,E1 270.802} C_DIS
LIN {X 0.233,Y -483.753,Z 291.502,A 0.000,B 0.000,C 90.000,E1 270.286} C_DIS
LIN {X -0.088,Y -482.837,Z 291.499,A 0.000,B 0.000,C 90.000,E1 269.828} C_DIS
LIN {X 0.069,Y -481.379,Z 291.496,A 0.000,B 0.000,C 90.000,E1 269.312} C_DIS
LIN {X 0.219,Y -479.334,Z 291.493,A 0.000,B 0.000,C 90.000,E1 268.797} C_DIS
LIN {X 0.050,Y -478.087,Z 291.492,A 0.000,B 0.000,C 90.000,E1 268.568} C_DIS
LIN {X 0.195,Y -474.955,Z 291.489,A 0.000,B 0.000,C 90.000,E1 268.051} C_DIS
LIN {X -0.166,Y -470.883,Z 291.487,A 0.000,B 0.000,C 90.000,E1 267.593} C_DIS
LIN {X 0.120,Y -468.449,Z 291.485,A 0.000,B 0.000,C 90.000,E1 267.306} C_DIS
LIN {X 0.228,Y -462.591,Z 291.482,A 0.000,B 0.000,C 90.000,E1 266.788} C_DIS
LIN {X -0.156,Y -459.510,Z 291.481,A 0.000,B 0.000,C 90.000,E1 266.617} C_DIS
LIN {X -0.114,Y -452.683,Z 291.479,A 0.000,B 0.000,C 90.000,E1 266.216} C_DIS
LIN {X -0.146,Y -448.959,Z 291.478,A 0.000,B 0.000,C 90.000,E1 266.045} C_DIS
LIN {X 0.119,Y -445.389,Z 291.477,A 0.000,B 0.000,C 90.000,E1 265.869} C_DIS
LIN {X -0.092,Y -440.929,Z 291.476,A 0.000,B 0.000,C 90.000,E1 265.755} C_DIS
LIN {X 0.029,Y -437.068,Z 291.476,A 0.000,B 0.000,C 90.000,E1 265.641} C_DIS
LIN {X 0.110,Y -427.904,Z 291.475,A 0.000,B 0.000,C 90.000,E1 265.469} C_DIS
LIN {X 0.073,Y -421.584,Z 291.475,A 0.000,B 0.000,C 90.000,E1 265.412} C_DIS
LIN {X -0.065,Y -415.519,Z 291.474,A 0.000,B 0.000,C 90.000,E1 265.412} C_DIS
LIN {X -0.059,Y -180.906,Z 291.474,A 0.000,B 0.000,C 90.000,E1 265.412} C_DIS
LIN {X 0.046,Y -180.677,Z 291.469,A 0.000,B 0.000,C 90.000,E1 264.489} C_DIS
LIN {X -0.055,Y -178.760,Z 291.441,A 0.000,B 0.000,C 90.000,E1 259.454} C_DIS
LIN {X 0.017,Y -175.807,Z 291.413,A 0.000,B 0.000,C 90.000,E1 254.338} C_DIS
LIN {X 0.011,Y -171.993,Z 291.385,A 0.000,B 0.000,C 90.000,E1 249.209} C_DIS
LIN {X 0.050,Y -171.404,Z 291.380,A 0.000,B 0.000,C 90.000,E1 248.337} C_DIS
LIN {X 0.034,Y -167.645,Z 291.356,A 0.000,B 0.000,C 90.000,E1 244.024} C_DIS
LIN {X 0.049,Y -166.306,Z 291.346,A 0.000,B 0.000,C 90.000,E1 242.281} C_DIS
LIN {X 0.042,Y -163.050,Z 291.327,A 0.000,B 0.000,C 90.000,E1 238.791} C_DIS
LIN {X 0.005,Y -160.984,Z 291.312,A 0.000,B 0.000,C 90.000,E1 236.167} C_DIS
LIN {X -0.018,Y -157.733,Z 291.292,A 0.000,B 0.000,C 90.000,E1 232.637} C_DIS
LIN {X -0.080,Y -155.771,Z 291.278,A 0.000,B 0.000,C 90.000,E1 229.989} C_DIS
LIN {X -0.024,Y -152.026,Z 291.253,A 0.000,B 0.000,C 90.000,E1 225.486} C_DIS
LIN {X -0.006,Y -150.274,Z 291.238,A 0.000,B 0.000,C 90.000,E1 222.771} C_DIS
LIN {X 0.011,Y -147.026,Z 291.212,A 0.000,B 0.000,C 90.000,E1 218.222} C_DIS
LIN {X 0.032,Y -145.608,Z 291.197,A 0.000,B 0.000,C 90.000,E1 215.471} C_DIS
LIN {X 0.035,Y -142.993,Z 291.172,A 0.000,B 0.000,C 90.000,E1 210.875} C_DIS
LIN {X -0.030,Y -141.620,Z 291.151,A 0.000,B 0.000,C 90.000,E1 207.206} C_DIS
LIN {X 0.027,Y -139.430,Z 291.115,A 0.000,B 0.000,C 90.000,E1 200.684} C_DIS
LIN {X -0.050,Y -139.161,Z 291.105,A 0.000,B 0.000,C 90.000,E1 198.852} C_DIS
LIN {X -0.012,Y -138.341,Z 291.058,A 0.000,B 0.000,C 90.000,E1 190.433} C_DIS
LIN {X -0.005,Y -139.479,Z 291.006,A 0.000,B 0.000,C 90.000,E1 181.088} C_DIS
LIN {X -0.065,Y -141.066,Z 290.975,A 0.000,B 0.000,C 90.000,E1 175.527} C_DIS
LIN {X 0.030,Y -142.440,Z 290.960,A 0.000,B 0.000,C 90.000,E1 172.704} C_DIS
LIN {X -0.020,Y -144.680,Z 290.934,A 0.000,B 0.000,C 90.000,E1 168.105} C_DIS
LIN {X 0.074,Y -147.269,Z 290.913,A 0.000,B 0.000,C 90.000,E1 164.393} C_DIS
LIN {X -0.051,Y -150.586,Z 290.888,A 0.000,B 0.000,C 90.000,E1 159.880} C_DIS
LIN {X 0.028,Y -154.058,Z 290.868,A 0.000,B 0.000,C 90.000,E1 156.230} C_DIS
LIN {X -0.046,Y -157.476,Z 290.848,A 0.000,B 0.000,C 90.000,E1 152.666} C_DIS
LIN {X 0.041,Y -161.700,Z 290.828,A 0.000,B 0.000,C 90.000,E1 149.076} C_DIS
LIN {X -0.082,Y -165.895,Z 290.809,A 0.000,B 0.000,C 90.000,E1 145.595} C_DIS
LIN {X 0.043,Y -170.877,Z 290.789,A 0.000,B 0.000,C 90.000,E1 142.065} C_DIS
LIN {X 0.070,Y -175.746,Z 290.770,A 0.000,B 0.000,C 90.000,E1 138.609} C_DIS
LIN {X -0.057,Y -181.356,Z 290.751,A 0.000,B 0.000,C 90.000,E1 135.243} C_DIS
LIN {X 0.078,Y -186.847,Z 290.733,A 0.000,B 0.000,C 90.000,E1 131.838} C_DIS
LIN {X 0.031,Y -191.434,Z 290.719,A 0.000,B 0.000,C 90.000,E1 129.358} C_DIS
LIN {X -0.036,Y -197.285,Z 290.700,A 0.000,B 0.000,C 90.000,E1 126.091} C_DIS
LIN {X 0.000,Y -200.563,Z 290.691,A 0.000,B 0.000,C 90.000,E1 124.452} C_DIS
LIN {X -0.013,Y -202.678,Z 290.685,A 0.000,B 0.000,C 90.000,E1 123.245} C_DIS
LIN {X -0.054,Y -303.968,Z 290.685,A 0.000,B 0.000,C 90.000,E1 123.245} C_DIS
LIN {X -0.064,Y -306.346,Z 290.684,A 0.000,B 0.000,C 90.000,E1 123.214} C_DIS
LIN {X -0.104,Y -310.432,Z 290.683,A 0.000,B 0.000,C 90.000,E1 123.038} C_DIS
LIN {X 0.027,Y -312.765,Z 290.682,A 0.000,B 0.000,C 90.000,E1 122.832} C_DIS
LIN {X 0.202,Y -316.625,Z 290.680,A 0.000,B 0.000,C 90.000,E1 122.339} C_DIS
LIN {X 0.014,Y -318.482,Z 290.678,A 0.000,B 0.000,C 90.000,E1 122.054} C_DIS
LIN {X -0.073,Y -319.932,Z 290.676,A 0.000,B 0.000,C 90.000,E1 121.750} C_DIS
LIN {X -0.009,Y -332.293,Z 290.659,A 0.000,B 0.000,C 90.000,E1 118.565} C_DIS
LIN {X -0.031,Y -344.883,Z 290.643,A 0.000,B 0.000,C 90.000,E1 115.771} C_DIS
LIN {X -0.027,Y -357.362,Z 290.630,A 0.000,B 0.000,C 90.000,E1 113.334} C_DIS
LIN {X 0.168,Y -371.148,Z 290.616,A 0.000,B 0.000,C 90.000,E1 110.918} C_DIS
LIN {X 0.097,Y -386.340,Z 290.603,A 0.000,B 0.000,C 90.000,E1 108.598} C_DIS
LIN {X 0.152,Y -403.052,Z 290.591,A 0.000,B 0.000,C 90.000,E1 106.315} C_DIS
LIN {X 0.004,Y -421.408,Z 290.578,A 0.000,B 0.000,C 90.000,E1 104.120} C_DIS
LIN {X -0.092,Y -441.248,Z 290.567,A 0.000,B 0.000,C 90.000,E1 102.007} C_DIS
LIN {X 0.191,Y -461.733,Z 290.556,A 0.000,B 0.000,C 90.000,E1 100.018} C_DIS
LIN {X -0.110,Y -485.395,Z 290.545,A 0.000,B 0.000,C 90.000,E1 98.049} C_DIS
LIN {X -0.004,Y -498.751,Z 290.539,A 0.000,B 0.000,C 90.000,E1 97.004} C_DIS
LIN {X 0.225,Y -500.949,Z 290.538,A 0.000,B 0.000,C 90.000,E1 96.777} C_DIS
LIN {X 0.216,Y -502.836,Z 290.537,A 0.000,B 0.000,C 90.000,E1 96.549} C_DIS
LIN {X -0.238,Y -504.272,Z 290.535,A 0.000,B 0.000,C 90.000,E1 96.372} C_DIS
LIN {X 0.065,Y -506.238,Z 290.533,A 0.000,B 0.000,C 90.000,E1 95.853} C_DIS
LIN {X -0.129,Y -507.056,Z 290.530,A 0.000,B 0.000,C 90.000,E1 95.391} C_DIS
LIN {X 0.149,Y -506.863,Z 290.527,A 0.000,B 0.000,C 90.000,E1 94.878} C_DIS
LIN {X -0.028,Y -505.626,Z 290.525,A 0.000,B 0.000,C 90.000,E1 94.416} C_DIS
LIN {X -0.137,Y -504.551,Z 290.523,A 0.000,B 0.000,C 90.000,E1 94.188} C_DIS
LIN {X -0.209,Y -503.096,Z 290.522,A 0.000,B 0.000,C 90.000,E1 93.955} C_DIS
LIN {X -0.055,Y -497.558,Z 290.518,A 0.000,B 0.000,C 90.000,E1 93.212} C_DIS
LIN {X -0.051,Y -489.552,Z 290.512,A 0.000,B 0.000,C 90.000,E1 92.236} C_DIS
LIN {X -0.228,Y -468.561,Z 290.499,A 0.000,B 0.000,C 90.000,E1 89.771} C_DIS
LIN {X -0.038,Y -453.060,Z 290.487,A 0.000,B 0.000,C 90.000,E1 87.707} C_DIS
LIN {X -0.084,Y -433.891,Z 290.471,A 0.000,B 0.000,C 90.000,E1 84.837} C_DIS
LIN {X 0.093,Y -418.080,Z 290.456,A 0.000,B 0.000,C 90.000,E1 82.129} C_DIS
LIN {X -0.009,Y -403.722,Z 290.441,A 0.000,B 0.000,C 90.000,E1 79.398} C_DIS
LIN {X 0.137,Y -395.099,Z 290.432,A 0.000,B 0.000,C 90.000,E1 77.701} C_DIS
LIN {X -0.120,Y -385.027,Z 290.421,A 0.000,B 0.000,C 90.000,E1 75.755} C_DIS
LIN {X -0.002,Y -373.605,Z 290.408,A 0.000,B 0.000,C 90.000,E1 73.433} C_DIS
LIN {X -0.057,Y -362.127,Z 290.395,A 0.000,B 0.000,C 90.000,E1 71.094} C_DIS
LIN {X -0.158,Y -350.855,Z 290.382,A 0.000,B 0.000,C 90.000,E1 68.720} C_DIS
LIN {X -0.001,Y -335.032,Z 290.361,A 0.000,B 0.000,C 90.000,E1 65.025} C_DIS
LIN {X 0.077,Y -322.117,Z 290.342,A 0.000,B 0.000,C 90.000,E1 61.563} C_DIS
LIN {X 0.136,Y -313.147,Z 290.328,A 0.000,B 0.000,C 90.000,E1 58.997} C_DIS
LIN {X -0.133,Y -302.492,Z 290.310,A 0.000,B 0.000,C 90.000,E1 55.801} C_DIS
LIN {X 0.031,Y -294.333,Z 290.295,A 0.000,B 0.000,C 90.000,E1 53.130} C_DIS
LIN {X 0.102,Y -286.216,Z 290.280,A 0.000,B 0.000,C 90.000,E1 50.436} C_DIS
LIN {X 0.108,Y -278.043,Z 290.265,A 0.000,B 0.000,C 90.000,E1 47.715} C_DIS
LIN {X 0.039,Y -268.295,Z 290.246,A 0.000,B 0.000,C 90.000,E1 44.271} C_DIS
LIN {X -0.025,Y -260.890,Z 290.230,A 0.000,B 0.000,C 90.000,E1 41.472} C_DIS
LIN {X 0.038,Y -255.290,Z 290.219,A 0.000,B 0.000,C 90.000,E1 39.322} C_DIS
LIN {X 0.063,Y -249.603,Z 290.207,A 0.000,B 0.000,C 90.000,E1 37.156} C_DIS
LIN {X 0.037,Y -243.673,Z 290.194,A 0.000,B 0.000,C 90.000,E1 34.978} C_DIS
LIN {X 0.119,Y -235.736,Z 290.178,A 0.000,B 0.000,C 90.000,E1 32.005} C_DIS
LIN {X 0.030,Y -228.324,Z 290.161,A 0.000,B 0.000,C 90.000,E1 29.027} C_DIS
LIN {X 0.049,Y -221.568,Z 290.144,A 0.000,B 0.000,C 90.000,E1 25.976} C_DIS
LIN {X 0.009,Y -215.555,Z 290.127,A 0.000,B 0.000,C 90.000,E1 22.898} C_DIS
LIN {X 0.054,Y -210.348,Z 290.110,A 0.000,B 0.000,C 90.000,E1 19.758} C_DIS
LIN {X -0.101,Y -204.776,Z 290.088,A 0.000,B 0.000,C 90.000,E1 15.843} C_DIS
LIN {X -0.054,Y -200.237,Z 290.066,A 0.000,B 0.000,C 90.000,E1 11.827} C_DIS
LIN {X 0.033,Y -196.145,Z 290.039,A 0.000,B 0.000,C 90.000,E1 6.947} C_DIS
LIN {X -0.056,Y -193.159,Z 290.007,A 0.000,B 0.000,C 90.000,E1 1.260} C_DIS
LIN {X -0.055,Y -194.290,Z 289.924,A 0.000,B 0.000,C 90.000,E1 346.408} C_DIS
LIN {X -0.058,Y -197.547,Z 289.897,A 0.000,B 0.000,C 90.000,E1 341.511} C_DIS
LIN {X 0.107,Y -201.505,Z 289.875,A 0.000,B 0.000,C 90.000,E1 337.411} C_DIS
LIN {X -0.034,Y -206.522,Z 289.852,A 0.000,B 0.000,C 90.000,E1 333.435} C_DIS
LIN {X -0.014,Y -212.437,Z 289.830,A 0.000,B 0.000,C 90.000,E1 329.459} C_DIS
LIN {X 0.083,Y -217.938,Z 289.813,A 0.000,B 0.000,C 90.000,E1 326.294} C_DIS
LIN {X 0.013,Y -224.244,Z 289.796,A 0.000,B 0.000,C 90.000,E1 323.210} C_DIS
LIN {X 0.010,Y -231.495,Z 289.779,A 0.000,B 0.000,C 90.000,E1 320.150} C_DIS
LIN {X -0.051,Y -240.795,Z 289.760,A 0.000,B 0.000,C 90.000,E1 316.782} C_DIS
LIN {X -0.028,Y -251.156,Z 289.741,A 0.000,B 0.000,C 90.000,E1 313.461} C_DIS
LIN {X -0.035,Y -262.500,Z 289.723,A 0.000,B 0.000,C 90.000,E1 310.216} C_DIS
LIN {X 0.022,Y -275.000,Z 289.706,A 0.000,B 0.000,C 90.000,E1 307.030} C_DIS
LIN {X 0.134,Y -288.936,Z 289.689,A 0.000,B 0.000,C 90.000,E1 303.913} C_DIS
LIN {X -0.033,Y -301.093,Z 289.675,A 0.000,B 0.000,C 90.000,E1 301.592} C_DIS
LIN {X 0.048,Y -320.348,Z 289.657,A 0.000,B 0.000,C 90.000,E1 298.309} C_DIS
LIN {X 0.045,Y -339.233,Z 289.642,A 0.000,B 0.000,C 90.000,E1 295.463} C_DIS
LIN {X -0.116,Y -352.197,Z 289.631,A 0.000,B 0.000,C 90.000,E1 293.643} C_DIS
LIN {X -0.113,Y -367.459,Z 289.620,A 0.000,B 0.000,C 90.000,E1 291.535} C_DIS
LIN {X 0.222,Y -385.130,Z 289.607,A 0.000,B 0.000,C 90.000,E1 289.141} C_DIS
LIN {X 0.023,Y -398.813,Z 289.597,A 0.000,B 0.000,C 90.000,E1 287.457} C_DIS
LIN {X -0.051,Y -412.356,Z 289.588,A 0.000,B 0.000,C 90.000,E1 285.788} C_DIS
LIN {X -0.022,Y -423.625,Z 289.580,A 0.000,B 0.000,C 90.000,E1 284.411} C_DIS
LIN {X 0.026,Y -430.164,Z 289.576,A 0.000,B 0.000,C 90.000,E1 283.592} C_DIS
LIN {X -0.090,Y -438.100,Z 289.570,A 0.000,B 0.000,C 90.000,E1 282.535} C_DIS
LIN {X -0.113,Y -445.357,Z 289.564,A 0.000,B 0.000,C 90.000,E1 281.478} C_DIS
LIN {X 0.115,Y -453.760,Z 289.556,A 0.000,B 0.000,C 90.000,E1 280.141} C_DIS
LIN {X 0.016,Y -461.421,Z 289.549,A 0.000,B 0.000,C 90.000,E1 278.859} C_DIS
LIN {X -0.042,Y -468.555,Z 289.542,A 0.000,B 0.000,C 90.000,E1 277.587} C_DIS
LIN {X 0.150,Y -473.920,Z 289.536,A 0.000,B 0.000,C 90.000,E1 276.549} C_DIS
LIN {X 0.123,Y -477.574,Z 289.532,A 0.000,B 0.000,C 90.000,E1 275.796} C_DIS
LIN {X -0.213,Y -479.773,Z 289.529,A 0.000,B 0.000,C 90.000,E1 275.334} C_DIS
LIN {X -0.102,Y -481.675,Z 289.527,A 0.000,B 0.000,C 90.000,E1 274.821} C_DIS
LIN {X 0.060,Y -483.170,Z 289.524,A 0.000,B 0.000,C 90.000,E1 274.302} C_DIS
LIN {X 0.229,Y -484.240,Z 289.521,A 0.000,B 0.000,C 90.000,E1 273.784} C_DIS
LIN {X -0.106,Y -484.938,Z 289.518,A 0.000,B 0.000,C 90.000,E1 273.326} C_DIS
LIN {X 0.075,Y -485.285,Z 289.516,A 0.000,B 0.000,C 90.000,E1 272.808} C_DIS
LIN {X 0.236,Y -485.317,Z 289.513,A 0.000,B 0.000,C 90.000,E1 272.293} C_DIS
LIN {X 0.097,Y -484.746,Z 289.507,A 0.000,B 0.000,C 90.000,E1 271.318} C_DIS
LIN {X -0.222,Y -484.350,Z 289.505,A 0.000,B 0.000,C 90.000,E1 270.859} C_DIS
LIN {X -0.059,Y -483.716,Z 289.502,A 0.000,B 0.000,C 90.000,E1 270.344} C_DIS
LIN {X 0.102,Y -482.783,Z 289.499,A 0.000,B 0.000,C 90.000,E1 269.828} C_DIS
LIN {X -0.223,Y -481.343,Z 289.496,A 0.000,B 0.000,C 90.000,E1 269.370} C_DIS
LIN {X -0.071,Y -479.346,Z 289.494,A 0.000,B 0.000,C 90.000,E1 268.854} C_DIS
LIN {X -0.239,Y -478.142,Z 289.492,A 0.000,B 0.000,C 90.000,E1 268.625} C_DIS
LIN {X -0.092,Y -475.078,Z 289.489,A 0.000,B 0.000,C 90.000,E1 268.108} C_DIS
LIN {X 0.020,Y -471.074,Z 289.487,A 0.000,B 0.000,C 90.000,E1 267.593} C_DIS
LIN {X -0.162,Y -468.696,Z 289.485,A 0.000,B 0.000,C 90.000,E1 267.364} C_DIS
LIN {X 0.109,Y -465.992,Z 289.484,A 0.000,B 0.000,C 90.000,E1 267.078} C_DIS
LIN {X -0.061,Y -462.948,Z 289.482,A 0.000,B 0.000,C 90.000,E1 266.846} C_DIS
LIN {X 0.008,Y -459.955,Z 289.481,A 0.000,B 0.000,C 90.000,E1 266.617} C_DIS
LIN {X 0.075,Y -456.522,Z 289.480,A 0.000,B 0.000,C 90.000,E1 266.388} C_DIS
LIN {X -0.014,Y -453.247,Z 289.479,A 0.000,B 0.000,C 90.000,E1 266.216} C_DIS
LIN {X -0.101,Y -449.460,Z 289.478,A 0.000,B 0.000,C 90.000,E1 266.045} C_DIS
LIN {X 0.143,Y -445.895,Z 289.477,A 0.000,B 0.000,C 90.000,E1 265.869} C_DIS
LIN {X -0.089,Y -441.522,Z 289.476,A 0.000,B 0.000,C 90.000,E1 265.755} C_DIS
LIN {X 0.094,Y -432.496,Z 289.475,A 0.000,B 0.000,C 90.000,E1 265.527} C_DIS
LIN {X 0.032,Y -428.371,Z 289.475,A 0.000,B 0.000,C 90.000,E1 265.469} C_DIS
LIN {X -0.028,Y -421.940,Z 289.474,A 0.000,B 0.000,C 90.000,E1 265.412} C_DIS
LIN {X -0.168,Y -417.541,Z 289.474,A 0.000,B 0.000,C 90.000,E1 265.412} C_DIS
LIN {X 0.076,Y -180.906,Z 289.474,A 0.000,B 0.000,C 90.000,E1 265.355} C_DIS
LIN {X -0.002,Y -180.669,Z 289.469,A 0.000,B 0.000,C 90.000,E1 264.489} C_DIS
LIN {X 0.073,Y -178.751,Z 289.441,A 0.000,B 0.000,C 90.000,E1 259.398} C_DIS
LIN {X -0.030,Y -175.797,Z 289.413,A 0.000,B 0.000,C 90.000,E1 254.338} C_DIS
LIN {X -0.036,Y -171.983,Z 289.384,A 0.000,B 0.000,C 90.000,E1 249.209} C_DIS
LIN {X 0.003,Y -171.389,Z 289.380,A 0.000,B 0.000,C 90.000,E1 248.337} C_DIS
LIN {X -0.012,Y -167.632,Z 289.356,A 0.000,B 0.000,C 90.000,E1 244.024} C_DIS
LIN {X 0.003,Y -166.289,Z 289.346,A 0.000,B 0.000,C 90.000,E1 242.281} C_DIS
LIN {X -0.003,Y -163.037,Z 289.327,A 0.000,B 0.000,C 90.000,E1 238.791} C_DIS
LIN {X -0.040,Y -160.967,Z 289.312,A 0.000,B 0.000,C 90.000,E1 236.167} C_DIS
LIN {X -0.063,Y -157.719,Z 289.292,A 0.000,B 0.000,C 90.000,E1 232.637} C_DIS
LIN {X 0.095,Y -155.759,Z 289.277,A 0.000,B 0.000,C 90.000,E1 229.908} C_DIS
LIN {X -0.067,Y -152.015,Z 289.253,A 0.000,B 0.000,C 90.000,E1 225.486} C_DIS
LIN {X -0.049,Y -150.262,Z 289.238,A 0.000,B 0.000,C 90.000,E1 222.771} C_DIS
LIN {X -0.031,Y -147.016,Z 289.212,A 0.000,B 0.000,C 90.000,E1 218.222} C_DIS
LIN {X -0.011,Y -145.599,Z 289.197,A 0.000,B 0.000,C 90.000,E1 215.471} C_DIS
LIN {X -0.006,Y -142.985,Z 289.172,A 0.000,B 0.000,C 90.000,E1 210.875} C_DIS
LIN {X -0.006,Y -141.612,Z 289.151,A 0.000,B 0.000,C 90.000,E1 207.180} C_DIS
LIN {X 0.035,Y -139.428,Z 289.115,A 0.000,B 0.000,C 90.000,E1 200.663} C_DIS
LIN {X -0.046,Y -139.157,Z 289.105,A 0.000,B 0.000,C 90.000,E1 198.833} C_DIS
LIN {X -0.028,Y -138.343,Z 289.058,A 0.000,B 0.000,C 90.000,E1 190.423} C_DIS
LIN {X -0.046,Y -139.481,Z 289.006,A 0.000,B 0.000,C 90.000,E1 181.088} C_DIS
LIN {X 0.034,Y -141.073,Z 288.975,A 0.000,B 0.000,C 90.000,E1 175.469} C_DIS
LIN {X -0.012,Y -142.449,Z 288.959,A 0.000,B 0.000,C 90.000,E1 172.704} C_DIS
LIN {X 0.078,Y -144.690,Z 288.934,A 0.000,B 0.000,C 90.000,E1 168.049} C_DIS
LIN {X 0.031,Y -147.282,Z 288.913,A 0.000,B 0.000,C 90.000,E1 164.393} C_DIS
LIN {X 0.048,Y -150.600,Z 288.888,A 0.000,B 0.000,C 90.000,E1 159.826} C_DIS
LIN {X -0.016,Y -154.074,Z 288.868,A 0.000,B 0.000,C 90.000,E1 156.230} C_DIS
LIN {X 0.049,Y -157.494,Z 288.848,A 0.000,B 0.000,C 90.000,E1 152.615} C_DIS
LIN {X -0.005,Y -161.722,Z 288.828,A 0.000,B 0.000,C 90.000,E1 149.076} C_DIS
LIN {X 0.009,Y -165.915,Z 288.809,A 0.000,B 0.000,C 90.000,E1 145.548} C_DIS
LIN {X -0.004,Y -170.901,Z 288.789,A 0.000,B 0.000,C 90.000,E1 142.065} C_DIS
LIN {X 0.023,Y -175.769,Z 288.770,A 0.000,B 0.000,C 90.000,E1 138.609} C_DIS
LIN {X 0.024,Y -181.378,Z 288.751,A 0.000,B 0.000,C 90.000,E1 135.202} C_DIS
LIN {X 0.027,Y -186.874,Z 288.732,A 0.000,B 0.000,C 90.000,E1 131.838} C_DIS
LIN {X -0.020,Y -191.457,Z 288.719,A 0.000,B 0.000,C 90.000,E1 129.358} C_DIS
LIN {X -0.088,Y -197.313,Z 288.700,A 0.000,B 0.000,C 90.000,E1 126.091} C_DIS
LIN {X -0.052,Y -200.591,Z 288.691,A 0.000,B 0.000,C 90.000,E1 124.452} C_DIS
LIN {X 0.097,Y -202.764,Z 288.684,A 0.000,B 0.000,C 90.000,E1 123.166} C_DIS
LIN {X 0.111,Y -304.711,Z 288.684,A 0.000,B 0.000,C 90.000,E1 123.166} C_DIS
LIN {X -0.015,Y -310.095,Z 288.683,A 0.000,B 0.000,C 90.000,E1 123.007} C_DIS
LIN {X -0.054,Y -312.571,Z 288.682,A 0.000,B 0.000,C 90.000,E1 122.832} C_DIS
LIN {X -0.187,Y -316.406,Z 288.680,A 0.000,B 0.000,C 90.000,E1 122.418} C_DIS
LIN {X -0.050,Y -318.290,Z 288.678,A 0.000,B 0.000,C 90.000,E1 122.084} C_DIS
LIN {X 0.088,Y -319.769,Z 288.676,A 0.000,B 0.000,C 90.000,E1 121.750} C_DIS
LIN {X -0.138,Y -332.153,Z 288.659,A 0.000,B 0.000,C 90.000,E1 118.615} C_DIS
LIN {X -0.017,Y -344.728,Z 288.643,A 0.000,B 0.000,C 90.000,E1 115.796} C_DIS
LIN {X 0.140,Y -357.193,Z 288.630,A 0.000,B 0.000,C 90.000,E1 113.334} C_DIS
LIN {X -0.009,Y -370.963,Z 288.617,A 0.000,B 0.000,C 90.000,E1 110.972} C_DIS
LIN {X -0.097,Y -386.139,Z 288.604,A 0.000,B 0.000,C 90.000,E1 108.652} C_DIS
LIN {X -0.061,Y -402.833,Z 288.591,A 0.000,B 0.000,C 90.000,E1 106.370} C_DIS
LIN {X 0.180,Y -421.170,Z 288.579,A 0.000,B 0.000,C 90.000,E1 104.120} C_DIS
LIN {X 0.080,Y -440.998,Z 288.567,A 0.000,B 0.000,C 90.000,E1 102.007} C_DIS
LIN {X -0.100,Y -461.478,Z 288.556,A 0.000,B 0.000,C 90.000,E1 100.074} C_DIS
LIN {X 0.046,Y -485.134,Z 288.545,A 0.000,B 0.000,C 90.000,E1 98.049} C_DIS
LIN {X 0.147,Y -498.498,Z 288.539,A 0.000,B 0.000,C 90.000,E1 97.004} C_DIS
LIN {X -0.123,Y -500.824,Z 288.538,A 0.000,B 0.000,C 90.000,E1 96.834} C_DIS
LIN {X -0.067,Y -502.742,Z 288.537,A 0.000,B 0.000,C 90.000,E1 96.606} C_DIS
LIN {X 0.049,Y -504.214,Z 288.535,A 0.000,B 0.000,C 90.000,E1 96.372} C_DIS
LIN {X -0.078,Y -505.437,Z 288.534,A 0.000,B 0.000,C 90.000,E1 96.144} C_DIS
LIN {X -0.152,Y -506.326,Z 288.533,A 0.000,B 0.000,C 90.000,E1 95.910} C_DIS
LIN {X 0.166,Y -507.258,Z 288.530,A 0.000,B 0.000,C 90.000,E1 95.391} C_DIS
LIN {X -0.062,Y -507.174,Z 288.527,A 0.000,B 0.000,C 90.000,E1 94.935} C_DIS
LIN {X -0.238,Y -506.055,Z 288.525,A 0.000,B 0.000,C 90.000,E1 94.473} C_DIS
LIN {X 0.158,Y -505.054,Z 288.523,A 0.000,B 0.000,C 90.000,E1 94.188} C_DIS
LIN {X 0.086,Y -503.688,Z 288.522,A 0.000,B 0.000,C 90.000,E1 93.955} C_DIS
LIN {X -0.256,Y -498.191,Z 288.518,A 0.000,B 0.000,C 90.000,E1 93.269} C_DIS
LIN {X -0.243,Y -490.239,Z 288.513,A 0.000,B 0.000,C 90.000,E1 92.293} C_DIS
LIN {X -0.030,Y -473.287,Z 288.502,A 0.000,B 0.000,C 90.000,E1 90.286} C_DIS
LIN {X 0.043,Y -455.513,Z 288.489,A 0.000,B 0.000,C 90.000,E1 87.993} C_DIS
LIN {X -0.129,Y -437.813,Z 288.474,A 0.000,B 0.000,C 90.000,E1 85.412} C_DIS
LIN {X 0.164,Y -421.638,Z 288.460,A 0.000,B 0.000,C 90.000,E1 82.704} C_DIS
LIN {X -0.085,Y -404.225,Z 288.441,A 0.000,B 0.000,C 90.000,E1 79.454} C_DIS
LIN {X 0.074,Y -395.604,Z 288.432,A 0.000,B 0.000,C 90.000,E1 77.757} C_DIS
LIN {X 0.205,Y -385.541,Z 288.421,A 0.000,B 0.000,C 90.000,E1 75.755} C_DIS
LIN {X -0.139,Y -374.128,Z 288.408,A 0.000,B 0.000,C 90.000,E1 73.504} C_DIS
LIN {X -0.148,Y -364.083,Z 288.397,A 0.000,B 0.000,C 90.000,E1 71.456} C_DIS
LIN {X 0.131,Y -352.794,Z 288.384,A 0.000,B 0.000,C 90.000,E1 69.028} C_DIS
LIN {X -0.102,Y -336.832,Z 288.363,A 0.000,B 0.000,C 90.000,E1 65.409} C_DIS
LIN {X -0.017,Y -322.635,Z 288.342,A 0.000,B 0.000,C 90.000,E1 61.641} C_DIS
LIN {X 0.051,Y -313.665,Z 288.328,A 0.000,B 0.000,C 90.000,E1 59.076} C_DIS
LIN {X -0.041,Y -303.007,Z 288.310,A 0.000,B 0.000,C 90.000,E1 55.849} C_DIS
LIN {X -0.035,Y -294.815,Z 288.296,A 0.000,B 0.000,C 90.000,E1 53.210} C_DIS
LIN {X 0.047,Y -286.688,Z 288.281,A 0.000,B 0.000,C 90.000,E1 50.517} C_DIS
LIN {X 0.066,Y -278.474,Z 288.266,A 0.000,B 0.000,C 90.000,E1 47.796} C_DIS
LIN {X 0.010,Y -268.704,Z 288.246,A 0.000,B 0.000,C 90.000,E1 44.352} C_DIS
LIN {X -0.042,Y -261.292,Z 288.231,A 0.000,B 0.000,C 90.000,E1 41.553} C_DIS
LIN {X 0.030,Y -255.701,Z 288.219,A 0.000,B 0.000,C 90.000,E1 39.402} C_DIS
LIN {X 0.063,Y -249.998,Z 288.207,A 0.000,B 0.000,C 90.000,E1 37.237} C_DIS
LIN {X -0.152,Y -244.109,Z 288.195,A 0.000,B 0.000,C 90.000,E1 35.105} C_DIS
LIN {X -0.057,Y -236.174,Z 288.178,A 0.000,B 0.000,C 90.000,E1 32.133} C_DIS
LIN {X -0.021,Y -228.748,Z 288.162,A 0.000,B 0.000,C 90.000,E1 29.127} C_DIS
LIN {X -0.098,Y -221.985,Z 288.145,A 0.000,B 0.000,C 90.000,E1 26.104} C_DIS
LIN {X -0.039,Y -215.955,Z 288.128,A 0.000,B 0.000,C 90.000,E1 23.003} C_DIS
LIN {X -0.063,Y -210.743,Z 288.110,A 0.000,B 0.000,C 90.000,E1 19.885} C_DIS
LIN {X 0.056,Y -205.132,Z 288.088,A 0.000,B 0.000,C 90.000,E1 15.898} C_DIS
LIN {X 0.065,Y -200.560,Z 288.066,A 0.000,B 0.000,C 90.000,E1 11.895} C_DIS
LIN {X -0.020,Y -196.435,Z 288.039,A 0.000,B 0.000,C 90.000,E1 7.068} C_DIS
LIN {X -0.075,Y -193.406,Z 288.008,A 0.000,B 0.000,C 90.000,E1 1.375} C_DIS
LIN {X -0.035,Y -194.462,Z 287.924,A 0.000,B 0.000,C 90.000,E1 346.408} C_DIS
LIN {X -0.032,Y -197.722,Z 287.897,A 0.000,B 0.000,C 90.000,E1 341.511} C_DIS
LIN {X -0.125,Y -201.658,Z 287.875,A 0.000,B 0.000,C 90.000,E1 337.486} C_DIS
LIN {X 0.004,Y -206.656,Z 287.852,A 0.000,B 0.000,C 90.000,E1 333.435} C_DIS
LIN {X 0.029,Y -212.554,Z 287.830,A 0.000,B 0.000,C 90.000,E1 329.459} C_DIS
LIN {X -0.052,Y -218.097,Z 287.813,A 0.000,B 0.000,C 90.000,E1 326.342} C_DIS
LIN {X 0.065,Y -224.425,Z 287.796,A 0.000,B 0.000,C 90.000,E1 323.210} C_DIS
LIN {X 0.070,Y -231.719,Z 287.779,A 0.000,B 0.000,C 90.000,E1 320.150} C_DIS
LIN {X 0.016,Y -241.011,Z 287.760,A 0.000,B 0.000,C 90.000,E1 316.782} C_DIS
LIN {X 0.048,Y -251.356,Z 287.742,A 0.000,B 0.000,C 90.000,E1 313.461} C_DIS
LIN {X -0.118,Y -262.691,Z 287.723,A 0.000,B 0.000,C 90.000,E1 310.253} C_DIS
LIN {X -0.102,Y -275.182,Z 287.706,A 0.000,B 0.000,C 90.000,E1 307.076} C_DIS
LIN {X -0.131,Y -287.503,Z 287.691,A 0.000,B 0.000,C 90.000,E1 304.326} C_DIS
LIN {X 0.082,Y -301.322,Z 287.676,A 0.000,B 0.000,C 90.000,E1 301.592} C_DIS
LIN {X -0.167,Y -318.558,Z 287.659,A 0.000,B 0.000,C 90.000,E1 298.693} C_DIS
LIN {X 0.060,Y -337.285,Z 287.643,A 0.000,B 0.000,C 90.000,E1 295.796} C_DIS
LIN {X 0.014,Y -350.232,Z 287.633,A 0.000,B 0.000,C 90.000,E1 293.951} C_DIS
LIN {X -0.018,Y -365.376,Z 287.621,A 0.000,B 0.000,C 90.000,E1 291.844} C_DIS
LIN {X 0.147,Y -380.739,Z 287.610,A 0.000,B 0.000,C 90.000,E1 289.758} C_DIS
LIN {X 0.038,Y -396.586,Z 287.599,A 0.000,B 0.000,C 90.000,E1 287.764} C_DIS
LIN {X -0.167,Y -407.841,Z 287.591,A 0.000,B 0.000,C 90.000,E1 286.386} C_DIS
LIN {X -0.077,Y -421.314,Z 287.582,A 0.000,B 0.000,C 90.000,E1 284.717} C_DIS
LIN {X 0.060,Y -427.917,Z 287.577,A 0.000,B 0.000,C 90.000,E1 283.883} C_DIS
LIN {X 0.152,Y -434.095,Z 287.573,A 0.000,B 0.000,C 90.000,E1 283.063} C_DIS
LIN {X 0.086,Y -441.660,Z 287.567,A 0.000,B 0.000,C 90.000,E1 282.007} C_DIS
LIN {X 0.105,Y -448.604,Z 287.561,A 0.000,B 0.000,C 90.000,E1 280.950} C_DIS
LIN {X 0.121,Y -455.130,Z 287.555,A 0.000,B 0.000,C 90.000,E1 279.905} C_DIS
LIN {X 0.043,Y -462.680,Z 287.548,A 0.000,B 0.000,C 90.000,E1 278.624} C_DIS
LIN {X -0.006,Y -469.718,Z 287.541,A 0.000,B 0.000,C 90.000,E1 277.352} C_DIS
LIN {X 0.197,Y -474.983,Z 287.535,A 0.000,B 0.000,C 90.000,E1 276.315} C_DIS
LIN {X -0.013,Y -479.570,Z 287.530,A 0.000,B 0.000,C 90.000,E1 275.334} C_DIS
LIN {X 0.098,Y -481.475,Z 287.527,A 0.000,B 0.000,C 90.000,E1 274.821} C_DIS
LIN {X -0.224,Y -482.973,Z 287.524,A 0.000,B 0.000,C 90.000,E1 274.359} C_DIS
LIN {X -0.055,Y -484.056,Z 287.521,A 0.000,B 0.000,C 90.000,E1 273.841} C_DIS
LIN {X 0.090,Y -484.744,Z 287.519,A 0.000,B 0.000,C 90.000,E1 273.326} C_DIS
LIN {X -0.213,Y -485.138,Z 287.516,A 0.000,B 0.000,C 90.000,E1 272.865} C_DIS
LIN {X -0.054,Y -485.180,Z 287.513,A 0.000,B 0.000,C 90.000,E1 272.350} C_DIS
LIN {X -0.194,Y -484.679,Z 287.508,A 0.000,B 0.000,C 90.000,E1 271.375} C_DIS
LIN {X 0.133,Y -483.676,Z 287.502,A 0.000,B 0.000,C 90.000,E1 270.344} C_DIS
LIN {X -0.189,Y -482.753,Z 287.499,A 0.000,B 0.000,C 90.000,E1 269.885} C_DIS
LIN {X -0.032,Y -481.337,Z 287.496,A 0.000,B 0.000,C 90.000,E1 269.370} C_DIS
LIN {X 0.119,Y -479.388,Z 287.494,A 0.000,B 0.000,C 90.000,E1 268.854} C_DIS
LIN {X -0.219,Y -476.764,Z 287.491,A 0.000,B 0.000,C 90.000,E1 268.396} C_DIS
LIN {X 0.095,Y -475.176,Z 287.490,A 0.000,B 0.000,C 90.000,E1 268.108} C_DIS
LIN {X 0.207,Y -471.271,Z 287.487,A 0.000,B 0.000,C 90.000,E1 267.593} C_DIS
LIN {X 0.023,Y -468.929,Z 287.485,A 0.000,B 0.000,C 90.000,E1 267.364} C_DIS
LIN {X 0.124,Y -463.293,Z 287.483,A 0.000,B 0.000,C 90.000,E1 266.846} C_DIS
LIN {X 0.162,Y -460.311,Z 287.481,A 0.000,B 0.000,C 90.000,E1 266.617} C_DIS
LIN {X 0.072,Y -453.722,Z 287.479,A 0.000,B 0.000,C 90.000,E1 266.216} C_DIS
LIN {X -0.050,Y -449.908,Z 287.478,A 0.000,B 0.000,C 90.000,E1 266.045} C_DIS
LIN {X 0.178,Y -446.393,Z 287.477,A 0.000,B 0.000,C 90.000,E1 265.869} C_DIS
LIN {X -0.071,Y -442.056,Z 287.476,A 0.000,B 0.000,C 90.000,E1 265.755} C_DIS
LIN {X 0.080,Y -433.390,Z 287.475,A 0.000,B 0.000,C 90.000,E1 265.527} C_DIS
LIN {X -0.084,Y -423.040,Z 287.474,A 0.000,B 0.000,C 90.000,E1 265.412} C_DIS
LIN {X 0.108,Y -416.729,Z 287.474,A 0.000,B 0.000,C 90.000,E1 265.355} C_DIS
LIN {X 0.014,Y -180.906,Z 287.474,A 0.000,B 0.000,C 90.000,E1 265.355} C_DIS
LIN {X -0.041,Y -180.663,Z 287.469,A 0.000,B 0.000,C 90.000,E1 264.489} C_DIS
LIN {X 0.034,Y -178.743,Z 287.441,A 0.000,B 0.000,C 90.000,E1 259.398} C_DIS
LIN {X -0.068,Y -175.791,Z 287.413,A 0.000,B 0.000,C 90.000,E1 254.338} C_DIS
LIN {X -0.073,Y -171.975,Z 287.384,A 0.000,B 0.000,C 90.000,E1 249.209} C_DIS
LIN {X -0.035,Y -171.378,Z 287.380,A 0.000,B 0.000,C 90.000,E1 248.337} C_DIS
LIN {X -0.050,Y -167.623,Z 287.356,A 0.000,B 0.000,C 90.000,E1 244.024} C_DIS
LIN {X -0.034,Y -166.276,Z 287.346,A 0.000,B 0.000,C 90.000,E1 242.281} C_DIS
LIN {X -0.040,Y -163.026,Z 287.327,A 0.000,B 0.000,C 90.000,E1 238.791} C_DIS
LIN {X 0.012,Y -160.953,Z 287.312,A 0.000,B 0.000,C 90.000,E1 236.135} C_DIS
LIN {X -0.004,Y -157.710,Z 287.292,A 0.000,B 0.000,C 90.000,E1 232.603} C_DIS
LIN {X 0.059,Y -155.749,Z 287.277,A 0.000,B 0.000,C 90.000,E1 229.908} C_DIS
LIN {X 0.005,Y -152.006,Z 287.252,A 0.000,B 0.000,C 90.000,E1 225.445} C_DIS
LIN {X -0.084,Y -150.251,Z 287.237,A 0.000,B 0.000,C 90.000,E1 222.771} C_DIS
LIN {X 0.050,Y -147.008,Z 287.212,A 0.000,B 0.000,C 90.000,E1 218.177} C_DIS
LIN {X 0.040,Y -145.591,Z 287.197,A 0.000,B 0.000,C 90.000,E1 215.438} C_DIS
LIN {X -0.041,Y -142.979,Z 287.171,A 0.000,B 0.000,C 90.000,E1 210.875} C_DIS
LIN {X -0.040,Y -141.606,Z 287.151,A 0.000,B 0.000,C 90.000,E1 207.180} C_DIS
LIN {X 0.001,Y -139.426,Z 287.115,A 0.000,B 0.000,C 90.000,E1 200.663} C_DIS
LIN {X 0.052,Y -139.154,Z 287.104,A 0.000,B 0.000,C 90.000,E1 198.779} C_DIS
LIN {X 0.075,Y -138.344,Z 287.058,A 0.000,B 0.000,C 90.000,E1 190.366} C_DIS
LIN {X 0.060,Y -139.484,Z 287.006,A 0.000,B 0.000,C 90.000,E1 181.031} C_DIS
LIN {X 0.001,Y -141.079,Z 286.975,A 0.000,B 0.000,C 90.000,E1 175.469} C_DIS
LIN {X -0.045,Y -142.455,Z 286.959,A 0.000,B 0.000,C 90.000,E1 172.704} C_DIS
LIN {X 0.044,Y -144.698,Z 286.934,A 0.000,B 0.000,C 90.000,E1 168.049} C_DIS
LIN {X -0.003,Y -147.292,Z 286.913,A 0.000,B 0.000,C 90.000,E1 164.393} C_DIS
LIN {X 0.012,Y -150.612,Z 286.888,A 0.000,B 0.000,C 90.000,E1 159.826} C_DIS
LIN {X -0.052,Y -154.087,Z 286.868,A 0.000,B 0.000,C 90.000,E1 156.230} C_DIS
LIN {X 0.014,Y -157.508,Z 286.848,A 0.000,B 0.000,C 90.000,E1 152.615} C_DIS
LIN {X -0.041,Y -161.738,Z 286.828,A 0.000,B 0.000,C 90.000,E1 149.076} C_DIS
LIN {X 0.065,Y -165.931,Z 286.809,A 0.000,B 0.000,C 90.000,E1 145.515} C_DIS
LIN {X -0.042,Y -170.920,Z 286.789,A 0.000,B 0.000,C 90.000,E1 142.065} C_DIS
LIN {X -0.016,Y -175.789,Z 286.770,A 0.000,B 0.000,C 90.000,E1 138.609} C_DIS
LIN {X -0.016,Y -181.398,Z 286.751,A 0.000,B 0.000,C 90.000,E1 135.202} C_DIS
LIN {X -0.012,Y -186.896,Z 286.732,A 0.000,B 0.000,C 90.000,E1 131.838} C_DIS
LIN {X -0.061,Y -191.478,Z 286.719,A 0.000,B 0.000,C 90.000,E1 129.358} C_DIS
LIN {X -0.129,Y -197.336,Z 286.700,A 0.000,B 0.000,C 90.000,E1 126.091} C_DIS
LIN {X 0.071,Y -200.613,Z 286.691,A 0.000,B 0.000,C 90.000,E1 124.405} C_DIS
LIN {X -0.053,Y -202.839,Z 286.684,A 0.000,B 0.000,C 90.000,E1 123.166} C_DIS
LIN {X -0.110,Y -304.588,Z 286.684,A 0.000,B 0.000,C 90.000,E1 123.166} C_DIS
LIN {X -0.203,Y -305.981,Z 286.684,A 0.000,B 0.000,C 90.000,E1 123.166} C_DIS
LIN {X 0.052,Y -310.101,Z 286.683,A 0.000,B 0.000,C 90.000,E1 122.959} C_DIS
LIN {X -0.118,Y -312.339,Z 286.682,A 0.000,B 0.000,C 90.000,E1 122.832} C_DIS
LIN {X -0.177,Y -316.218,Z 286.680,A 0.000,B 0.000,C 90.000,E1 122.418} C_DIS
LIN {X 0.013,Y -318.123,Z 286.678,A 0.000,B 0.000,C 90.000,E1 122.084} C_DIS
LIN {X -0.066,Y -319.623,Z 286.677,A 0.000,B 0.000,C 90.000,E1 121.799} C_DIS
LIN {X -0.061,Y -333.369,Z 286.657,A 0.000,B 0.000,C 90.000,E1 118.309} C_DIS
LIN {X -0.059,Y -346.100,Z 286.642,A 0.000,B 0.000,C 90.000,E1 115.515} C_DIS
LIN {X -0.025,Y -358.714,Z 286.628,A 0.000,B 0.000,C 90.000,E1 113.078} C_DIS
LIN {X 0.069,Y -372.643,Z 286.615,A 0.000,B 0.000,C 90.000,E1 110.684} C_DIS
LIN {X 0.036,Y -387.991,Z 286.602,A 0.000,B 0.000,C 90.000,E1 108.362} C_DIS
LIN {X 0.135,Y -404.871,Z 286.589,A 0.000,B 0.000,C 90.000,E1 106.079} C_DIS
LIN {X 0.032,Y -423.409,Z 286.577,A 0.000,B 0.000,C 90.000,E1 103.883} C_DIS
LIN {X 0.054,Y -443.355,Z 286.565,A 0.000,B 0.000,C 90.000,E1 101.771} C_DIS
LIN {X -0.050,Y -463.898,Z 286.555,A 0.000,B 0.000,C 90.000,E1 99.849} C_DIS
LIN {X -0.117,Y -487.587,Z 286.544,A 0.000,B 0.000,C 90.000,E1 97.871} C_DIS
LIN {X 0.193,Y -498.302,Z 286.539,A 0.000,B 0.000,C 90.000,E1 97.011} C_DIS
LIN {X -0.017,Y -500.734,Z 286.538,A 0.000,B 0.000,C 90.000,E1 96.834} C_DIS
LIN {X -0.237,Y -504.186,Z 286.536,A 0.000,B 0.000,C 90.000,E1 96.429} C_DIS
LIN {X 0.133,Y -505.480,Z 286.534,A 0.000,B 0.000,C 90.000,E1 96.144} C_DIS
LIN {X 0.054,Y -506.427,Z 286.533,A 0.000,B 0.000,C 90.000,E1 95.910} C_DIS
LIN {X -0.133,Y -507.452,Z 286.530,A 0.000,B 0.000,C 90.000,E1 95.448} C_DIS
LIN {X 0.145,Y -507.454,Z 286.527,A 0.000,B 0.000,C 90.000,E1 94.935} C_DIS
LIN {X -0.031,Y -506.429,Z 286.525,A 0.000,B 0.000,C 90.000,E1 94.473} C_DIS
LIN {X -0.138,Y -505.482,Z 286.523,A 0.000,B 0.000,C 90.000,E1 94.245} C_DIS
LIN {X -0.209,Y -504.186,Z 286.522,A 0.000,B 0.000,C 90.000,E1 94.012} C_DIS
LIN {X -0.047,Y -498.769,Z 286.518,A 0.000,B 0.000,C 90.000,E1 93.269} C_DIS
LIN {X -0.030,Y -490.824,Z 286.513,A 0.000,B 0.000,C 90.000,E1 92.293} C_DIS
LIN {X 0.054,Y -478.034,Z 286.504,A 0.000,B 0.000,C 90.000,E1 90.802} C_DIS
LIN {X -0.230,Y -459.834,Z 286.492,A 0.000,B 0.000,C 90.000,E1 88.568} C_DIS
LIN {X -0.029,Y -443.436,Z 286.479,A 0.000,B 0.000,C 90.000,E1 86.216} C_DIS
LIN {X 0.126,Y -425.197,Z 286.463,A 0.000,B 0.000,C 90.000,E1 83.280} C_DIS
LIN {X 0.040,Y -411.723,Z 286.449,A 0.000,B 0.000,C 90.000,E1 80.849} C_DIS
LIN {X -0.036,Y -401.841,Z 286.438,A 0.000,B 0.000,C 90.000,E1 78.926} C_DIS
LIN {X -0.173,Y -390.319,Z 286.426,A 0.000,B 0.000,C 90.000,E1 76.700} C_DIS
LIN {X -0.027,Y -378.864,Z 286.413,A 0.000,B 0.000,C 90.000,E1 74.393} C_DIS
LIN {X -0.036,Y -370.276,Z 286.404,A 0.000,B 0.000,C 90.000,E1 72.653} C_DIS
LIN {X -0.054,Y -358.889,Z 286.390,A 0.000,B 0.000,C 90.000,E1 70.296} C_DIS
LIN {X -0.043,Y -345.102,Z 286.374,A 0.000,B 0.000,C 90.000,E1 67.283} C_DIS
LIN {X 0.054,Y -330.013,Z 286.353,A 0.000,B 0.000,C 90.000,E1 63.563} C_DIS
LIN {X 0.021,Y -318.626,Z 286.336,A 0.000,B 0.000,C 90.000,E1 60.411} C_DIS
LIN {X -0.015,Y -307.654,Z 286.318,A 0.000,B 0.000,C 90.000,E1 57.199} C_DIS
LIN {X 0.098,Y -299.348,Z 286.303,A 0.000,B 0.000,C 90.000,E1 54.562} C_DIS
LIN {X 0.111,Y -291.171,Z 286.288,A 0.000,B 0.000,C 90.000,E1 51.904} C_DIS
LIN {X 0.001,Y -285.058,Z 286.277,A 0.000,B 0.000,C 90.000,E1 49.908} C_DIS
LIN {X -0.019,Y -276.871,Z 286.262,A 0.000,B 0.000,C 90.000,E1 47.187} C_DIS
LIN {X 0.064,Y -267.212,Z 286.243,A 0.000,B 0.000,C 90.000,E1 43.704} C_DIS
LIN {X -0.033,Y -259.796,Z 286.227,A 0.000,B 0.000,C 90.000,E1 40.906} C_DIS
LIN {X 0.039,Y -254.204,Z 286.215,A 0.000,B 0.000,C 90.000,E1 38.749} C_DIS
LIN {X 0.046,Y -248.457,Z 286.203,A 0.000,B 0.000,C 90.000,E1 36.583} C_DIS
LIN {X -0.001,Y -242.511,Z 286.191,A 0.000,B 0.000,C 90.000,E1 34.405} C_DIS
LIN {X -0.081,Y -232.770,Z 286.171,A 0.000,B 0.000,C 90.000,E1 30.718} C_DIS
LIN {X -0.046,Y -225.652,Z 286.154,A 0.000,B 0.000,C 90.000,E1 27.692} C_DIS
LIN {X -0.098,Y -219.284,Z 286.137,A 0.000,B 0.000,C 90.000,E1 24.643} C_DIS
LIN {X -0.078,Y -213.633,Z 286.120,A 0.000,B 0.000,C 90.000,E1 21.535} C_DIS
LIN {X 0.004,Y -207.608,Z 286.098,A 0.000,B 0.000,C 90.000,E1 17.583} C_DIS
LIN {X 0.045,Y -202.593,Z 286.076,A 0.000,B 0.000,C 90.000,E1 13.592} C_DIS
LIN {X 0.090,Y -198.621,Z 286.053,A 0.000,B 0.000,C 90.000,E1 9.557} C_DIS
LIN {X 0.037,Y -195.151,Z 286.026,A 0.000,B 0.000,C 90.000,E1 4.702} C_DIS
LIN {X 0.041,Y -192.644,Z 285.988,A 0.000,B 0.000,C 90.000,E1 357.879} C_DIS
LIN {X -0.021,Y -194.218,Z 285.929,A 0.000,B 0.000,C 90.000,E1 347.229} C_DIS
LIN {X 0.051,Y -197.228,Z 285.902,A 0.000,B 0.000,C 90.000,E1 342.308} C_DIS
LIN {X -0.060,Y -200.956,Z 285.879,A 0.000,B 0.000,C 90.000,E1 338.284} C_DIS
LIN {X 0.060,Y -205.711,Z 285.857,A 0.000,B 0.000,C 90.000,E1 334.229} C_DIS
LIN {X 0.047,Y -211.436,Z 285.835,A 0.000,B 0.000,C 90.000,E1 330.255} C_DIS
LIN {X 0.005,Y -216.802,Z 285.817,A 0.000,B 0.000,C 90.000,E1 327.120} C_DIS
LIN {X 0.087,Y -222.935,Z 285.800,A 0.000,B 0.000,C 90.000,E1 323.989} C_DIS
LIN {X -0.087,Y -230.031,Z 285.783,A 0.000,B 0.000,C 90.000,E1 320.964} C_DIS
LIN {X -0.022,Y -239.086,Z 285.764,A 0.000,B 0.000,C 90.000,E1 317.553} C_DIS
LIN {X 0.131,Y -249.157,Z 285.746,A 0.000,B 0.000,C 90.000,E1 314.190} C_DIS
LIN {X -0.115,Y -260.282,Z 285.728,A 0.000,B 0.000,C 90.000,E1 310.987} C_DIS
LIN {X -0.173,Y -272.476,Z 285.710,A 0.000,B 0.000,C 90.000,E1 307.810} C_DIS
LIN {X -0.107,Y -284.507,Z 285.694,A 0.000,B 0.000,C 90.000,E1 305.025} C_DIS
LIN {X 0.035,Y -296.180,Z 285.681,A 0.000,B 0.000,C 90.000,E1 302.625} C_DIS
LIN {X -0.052,Y -312.881,Z 285.665,A 0.000,B 0.000,C 90.000,E1 299.667} C_DIS
LIN {X -0.179,Y -333.254,Z 285.647,A 0.000,B 0.000,C 90.000,E1 296.488} C_DIS
LIN {X 0.002,Y -346.116,Z 285.637,A 0.000,B 0.000,C 90.000,E1 294.591} C_DIS
LIN {X -0.029,Y -359.009,Z 285.626,A 0.000,B 0.000,C 90.000,E1 292.770} C_DIS
LIN {X 0.131,Y -374.232,Z 285.615,A 0.000,B 0.000,C 90.000,E1 290.663} C_DIS
LIN {X 0.021,Y -392.088,Z 285.602,A 0.000,B 0.000,C 90.000,E1 288.362} C_DIS
LIN {X -0.058,Y -405.587,Z 285.593,A 0.000,B 0.000,C 90.000,E1 286.677} C_DIS
LIN {X 0.116,Y -421.248,Z 285.582,A 0.000,B 0.000,C 90.000,E1 284.717} C_DIS
LIN {X -0.158,Y -427.838,Z 285.577,A 0.000,B 0.000,C 90.000,E1 283.939} C_DIS
LIN {X -0.073,Y -433.969,Z 285.573,A 0.000,B 0.000,C 90.000,E1 283.119} C_DIS
LIN {X 0.082,Y -439.673,Z 285.568,A 0.000,B 0.000,C 90.000,E1 282.299} C_DIS
LIN {X 0.078,Y -446.740,Z 285.563,A 0.000,B 0.000,C 90.000,E1 281.243} C_DIS
LIN {X 0.071,Y -453.349,Z 285.557,A 0.000,B 0.000,C 90.000,E1 280.197} C_DIS
LIN {X -0.036,Y -461.021,Z 285.549,A 0.000,B 0.000,C 90.000,E1 278.916} C_DIS
LIN {X 0.124,Y -466.757,Z 285.544,A 0.000,B 0.000,C 90.000,E1 277.871} C_DIS
LIN {X 0.082,Y -473.494,Z 285.537,A 0.000,B 0.000,C 90.000,E1 276.606} C_DIS
LIN {X 0.051,Y -477.184,Z 285.533,A 0.000,B 0.000,C 90.000,E1 275.853} C_DIS
LIN {X 0.189,Y -479.365,Z 285.530,A 0.000,B 0.000,C 90.000,E1 275.334} C_DIS
LIN {X -0.181,Y -481.264,Z 285.527,A 0.000,B 0.000,C 90.000,E1 274.878} C_DIS
LIN {X -0.022,Y -482.767,Z 285.524,A 0.000,B 0.000,C 90.000,E1 274.359} C_DIS
LIN {X 0.145,Y -483.864,Z 285.521,A 0.000,B 0.000,C 90.000,E1 273.841} C_DIS
LIN {X -0.194,Y -484.600,Z 285.519,A 0.000,B 0.000,C 90.000,E1 273.383} C_DIS
LIN {X -0.015,Y -484.984,Z 285.516,A 0.000,B 0.000,C 90.000,E1 272.865} C_DIS
LIN {X 0.144,Y -485.044,Z 285.513,A 0.000,B 0.000,C 90.000,E1 272.350} C_DIS
LIN {X 0.002,Y -484.595,Z 285.508,A 0.000,B 0.000,C 90.000,E1 271.375} C_DIS
LIN {X 0.165,Y -484.197,Z 285.505,A 0.000,B 0.000,C 90.000,E1 270.859} C_DIS
LIN {X -0.156,Y -483.619,Z 285.502,A 0.000,B 0.000,C 90.000,E1 270.401} C_DIS
LIN {X 0.004,Y -482.722,Z 285.499,A 0.000,B 0.000,C 90.000,E1 269.885} C_DIS
LIN {X 0.162,Y -481.347,Z 285.497,A 0.000,B 0.000,C 90.000,E1 269.370} C_DIS
LIN {X -0.169,Y -479.423,Z 285.494,A 0.000,B 0.000,C 90.000,E1 268.912} C_DIS
LIN {X -0.028,Y -476.860,Z 285.491,A 0.000,B 0.000,C 90.000,E1 268.396} C_DIS
LIN {X 0.109,Y -473.473,Z 285.488,A 0.000,B 0.000,C 90.000,E1 267.879} C_DIS
LIN {X -0.074,Y -471.459,Z 285.487,A 0.000,B 0.000,C 90.000,E1 267.650} C_DIS
LIN {X 0.016,Y -466.565,Z 285.484,A 0.000,B 0.000,C 90.000,E1 267.135} C_DIS
LIN {X -0.177,Y -463.706,Z 285.483,A 0.000,B 0.000,C 90.000,E1 266.906} C_DIS
LIN {X -0.157,Y -460.739,Z 285.481,A 0.000,B 0.000,C 90.000,E1 266.674} C_DIS
LIN {X 0.157,Y -454.189,Z 285.479,A 0.000,B 0.000,C 90.000,E1 266.216} C_DIS
LIN {X 0.223,Y -447.021,Z 285.477,A 0.000,B 0.000,C 90.000,E1 265.869} C_DIS
LIN {X 0.004,Y -439.036,Z 285.476,A 0.000,B 0.000,C 90.000,E1 265.641} C_DIS
LIN {X -0.035,Y -430.090,Z 285.475,A 0.000,B 0.000,C 90.000,E1 265.469} C_DIS
LIN {X 0.134,Y -421.898,Z 285.474,A 0.000,B 0.000,C 90.000,E1 265.355} C_DIS
LIN {X -0.023,Y -416.399,Z 285.474,A 0.000,B 0.000,C 90.000,E1 265.355} C_DIS
LIN {X -0.044,Y -180.906,Z 285.474,A 0.000,B 0.000,C 90.000,E1 265.355} C_DIS
LIN {X -0.073,Y -180.658,Z 285.469,A 0.000,B 0.000,C 90.000,E1 264.489} C_DIS
LIN {X 0.003,Y -178.738,Z 285.441,A 0.000,B 0.000,C 90.000,E1 259.398} C_DIS
LIN {X 0.070,Y -175.786,Z 285.413,A 0.000,B 0.000,C 90.000,E1 254.283} C_DIS
LIN {X 0.058,Y -171.970,Z 285.384,A 0.000,B 0.000,C 90.000,E1 249.156} C_DIS
LIN {X -0.065,Y -171.369,Z 285.380,A 0.000,B 0.000,C 90.000,E1 248.337} C_DIS
LIN {X -0.079,Y -167.616,Z 285.356,A 0.000,B 0.000,C 90.000,E1 244.024} C_DIS
LIN {X -0.064,Y -166.266,Z 285.346,A 0.000,B 0.000,C 90.000,E1 242.281} C_DIS
LIN {X 0.071,Y -163.018,Z 285.326,A 0.000,B 0.000,C 90.000,E1 238.742} C_DIS
LIN {X -0.016,Y -160.943,Z 285.312,A 0.000,B 0.000,C 90.000,E1 236.135} C_DIS
LIN {X -0.032,Y -157.701,Z 285.292,A 0.000,B 0.000,C 90.000,E1 232.603} C_DIS
LIN {X 0.031,Y -155.741,Z 285.277,A 0.000,B 0.000,C 90.000,E1 229.908} C_DIS
LIN {X 0.084,Y -151.998,Z 285.252,A 0.000,B 0.000,C 90.000,E1 225.405} C_DIS
LIN {X -0.010,Y -150.243,Z 285.237,A 0.000,B 0.000,C 90.000,E1 222.732} C_DIS
LIN {X 0.023,Y -147.002,Z 285.212,A 0.000,B 0.000,C 90.000,E1 218.177} C_DIS
LIN {X 0.013,Y -145.586,Z 285.197,A 0.000,B 0.000,C 90.000,E1 215.438} C_DIS
LIN {X 0.007,Y -142.974,Z 285.171,A 0.000,B 0.000,C 90.000,E1 210.846} C_DIS
LIN {X 0.060,Y -141.601,Z 285.151,A 0.000,B 0.000,C 90.000,E1 207.129} C_DIS
LIN {X -0.025,Y -139.423,Z 285.115,A 0.000,B 0.000,C 90.000,E1 200.663} C_DIS
LIN {X 0.026,Y -139.152,Z 285.104,A 0.000,B 0.000,C 90.000,E1 198.779} C_DIS
LIN {X 0.048,Y -138.345,Z 285.058,A 0.000,B 0.000,C 90.000,E1 190.366} C_DIS
LIN {X 0.034,Y -139.485,Z 285.006,A 0.000,B 0.000,C 90.000,E1 181.031} C_DIS
LIN {X -0.026,Y -141.084,Z 284.975,A 0.000,B 0.000,C 90.000,E1 175.469} C_DIS
LIN {X -0.072,Y -142.460,Z 284.959,A 0.000,B 0.000,C 90.000,E1 172.704} C_DIS
LIN {X 0.017,Y -144.704,Z 284.934,A 0.000,B 0.000,C 90.000,E1 168.049} C_DIS
LIN {X -0.031,Y -147.301,Z 284.913,A 0.000,B 0.000,C 90.000,E1 164.393} C_DIS
LIN {X -0.015,Y -150.621,Z 284.888,A 0.000,B 0.000,C 90.000,E1 159.826} C_DIS
LIN {X 0.061,Y -154.097,Z 284.868,A 0.000,B 0.000,C 90.000,E1 156.177} C_DIS
LIN {X -0.015,Y -157.519,Z 284.848,A 0.000,B 0.000,C 90.000,E1 152.615} C_DIS
LIN {X -0.070,Y -161.752,Z 284.828,A 0.000,B 0.000,C 90.000,E1 149.076} C_DIS
LIN {X 0.036,Y -165.945,Z 284.808,A 0.000,B 0.000,C 90.000,E1 145.515} C_DIS
LIN {X 0.033,Y -170.936,Z 284.789,A 0.000,B 0.000,C 90.000,E1 142.029} C_DIS
LIN {X -0.047,Y -175.804,Z 284.770,A 0.000,B 0.000,C 90.000,E1 138.609} C_DIS
LIN {X 0.081,Y -181.412,Z 284.751,A 0.000,B 0.000,C 90.000,E1 135.162} C_DIS
LIN {X -0.044,Y -186.914,Z 284.732,A 0.000,B 0.000,C 90.000,E1 131.838} C_DIS
LIN {X 0.029,Y -191.493,Z 284.719,A 0.000,B 0.000,C 90.000,E1 129.322} C_DIS
LIN {X 0.114,Y -197.355,Z 284.700,A 0.000,B 0.000,C 90.000,E1 126.011} C_DIS
LIN {X 0.039,Y -200.631,Z 284.691,A 0.000,B 0.000,C 90.000,E1 124.405} C_DIS
LIN {X 0.074,Y -202.916,Z 284.684,A 0.000,B 0.000,C 90.000,E1 123.086} C_DIS
LIN {X 0.057,Y -304.989,Z 284.684,A 0.000,B 0.000,C 90.000,E1 123.086} C_DIS
LIN {X -0.052,Y -306.352,Z 284.684,A 0.000,B 0.000,C 90.000,E1 123.086} C_DIS
LIN {X 0.000,Y -312.019,Z 284.682,A 0.000,B 0.000,C 90.000,E1 122.801} C_DIS
LIN {X 0.009,Y -315.120,Z 284.681,A 0.000,B 0.000,C 90.000,E1 122.498} C_DIS
LIN {X 0.130,Y -318.757,Z 284.677,A 0.000,B 0.000,C 90.000,E1 121.926} C_DIS
LIN {X 0.029,Y -320.252,Z 284.676,A 0.000,B 0.000,C 90.000,E1 121.623} C_DIS
LIN {X 0.103,Y -332.684,Z 284.658,A 0.000,B 0.000,C 90.000,E1 118.437} C_DIS
LIN {X -0.057,Y -345.334,Z 284.643,A 0.000,B 0.000,C 90.000,E1 115.668} C_DIS
LIN {X 0.112,Y -357.868,Z 284.629,A 0.000,B 0.000,C 90.000,E1 113.206} C_DIS
LIN {X -0.023,Y -371.712,Z 284.616,A 0.000,B 0.000,C 90.000,E1 110.844} C_DIS
LIN {X 0.145,Y -386.968,Z 284.603,A 0.000,B 0.000,C 90.000,E1 108.489} C_DIS
LIN {X -0.160,Y -403.748,Z 284.590,A 0.000,B 0.000,C 90.000,E1 106.260} C_DIS
LIN {X 0.108,Y -422.180,Z 284.578,A 0.000,B 0.000,C 90.000,E1 104.008} C_DIS
LIN {X 0.068,Y -442.069,Z 284.566,A 0.000,B 0.000,C 90.000,E1 101.895} C_DIS
LIN {X -0.032,Y -462.578,Z 284.555,A 0.000,B 0.000,C 90.000,E1 99.962} C_DIS
LIN {X -0.260,Y -486.236,Z 284.544,A 0.000,B 0.000,C 90.000,E1 97.992} C_DIS
LIN {X -0.145,Y -499.619,Z 284.539,A 0.000,B 0.000,C 90.000,E1 96.947} C_DIS
LIN {X -0.140,Y -503.452,Z 284.536,A 0.000,B 0.000,C 90.000,E1 96.543} C_DIS
LIN {X 0.224,Y -504.990,Z 284.535,A 0.000,B 0.000,C 90.000,E1 96.258} C_DIS
LIN {X 0.089,Y -506.137,Z 284.534,A 0.000,B 0.000,C 90.000,E1 96.030} C_DIS
LIN {X -0.096,Y -507.491,Z 284.531,A 0.000,B 0.000,C 90.000,E1 95.568} C_DIS
LIN {X 0.228,Y -507.792,Z 284.528,A 0.000,B 0.000,C 90.000,E1 95.049} C_DIS
LIN {X 0.052,Y -507.083,Z 284.526,A 0.000,B 0.000,C 90.000,E1 94.588} C_DIS
LIN {X -0.161,Y -505.239,Z 284.523,A 0.000,B 0.000,C 90.000,E1 94.131} C_DIS
LIN {X -0.234,Y -503.775,Z 284.522,A 0.000,B 0.000,C 90.000,E1 93.898} C_DIS
LIN {X -0.163,Y -496.294,Z 284.516,A 0.000,B 0.000,C 90.000,E1 92.922} C_DIS
LIN {X -0.195,Y -488.080,Z 284.511,A 0.000,B 0.000,C 90.000,E1 91.949} C_DIS
LIN {X -0.129,Y -465.096,Z 284.495,A 0.000,B 0.000,C 90.000,E1 89.198} C_DIS
LIN {X 0.208,Y -451.802,Z 284.486,A 0.000,B 0.000,C 90.000,E1 87.364} C_DIS
LIN {X -0.048,Y -434.435,Z 284.471,A 0.000,B 0.000,C 90.000,E1 84.780} C_DIS
LIN {X 0.199,Y -418.608,Z 284.456,A 0.000,B 0.000,C 90.000,E1 82.064} C_DIS
LIN {X 0.049,Y -404.275,Z 284.441,A 0.000,B 0.000,C 90.000,E1 79.342} C_DIS
LIN {X -0.186,Y -395.650,Z 284.432,A 0.000,B 0.000,C 90.000,E1 77.701} C_DIS
LIN {X -0.045,Y -385.611,Z 284.421,A 0.000,B 0.000,C 90.000,E1 75.700} C_DIS
LIN {X -0.032,Y -375.661,Z 284.409,A 0.000,B 0.000,C 90.000,E1 73.685} C_DIS
LIN {X 0.070,Y -364.216,Z 284.396,A 0.000,B 0.000,C 90.000,E1 71.329} C_DIS
LIN {X 0.069,Y -351.581,Z 284.381,A 0.000,B 0.000,C 90.000,E1 68.646} C_DIS
LIN {X 0.114,Y -335.888,Z 284.361,A 0.000,B 0.000,C 90.000,E1 64.973} C_DIS
LIN {X -0.137,Y -321.820,Z 284.340,A 0.000,B 0.000,C 90.000,E1 61.257} C_DIS
LIN {X 0.071,Y -312.888,Z 284.326,A 0.000,B 0.000,C 90.000,E1 58.663} C_DIS
LIN {X -0.034,Y -302.309,Z 284.308,A 0.000,B 0.000,C 90.000,E1 55.435} C_DIS
LIN {X 0.127,Y -294.089,Z 284.293,A 0.000,B 0.000,C 90.000,E1 52.763} C_DIS
LIN {X -0.031,Y -285.925,Z 284.278,A 0.000,B 0.000,C 90.000,E1 50.114} C_DIS
LIN {X -0.023,Y -277.684,Z 284.263,A 0.000,B 0.000,C 90.000,E1 47.391} C_DIS
LIN {X -0.097,Y -267.979,Z 284.244,A 0.000,B 0.000,C 90.000,E1 43.947} C_DIS
LIN {X -0.167,Y -260.563,Z 284.228,A 0.000,B 0.000,C 90.000,E1 41.148} C_DIS
LIN {X -0.076,Y -254.986,Z 284.217,A 0.000,B 0.000,C 90.000,E1 38.991} C_DIS
LIN {X 0.101,Y -249.248,Z 284.205,A 0.000,B 0.000,C 90.000,E1 36.790} C_DIS
LIN {X 0.067,Y -243.326,Z 284.192,A 0.000,B 0.000,C 90.000,E1 34.612} C_DIS
LIN {X 0.010,Y -233.558,Z 284.172,A 0.000,B 0.000,C 90.000,E1 30.924} C_DIS
LIN {X 0.065,Y -226.408,Z 284.155,A 0.000,B 0.000,C 90.000,E1 27.897} C_DIS
LIN {X 0.033,Y -219.978,Z 284.138,A 0.000,B 0.000,C 90.000,E1 24.847} C_DIS
LIN {X -0.045,Y -214.315,Z 284.121,A 0.000,B 0.000,C 90.000,E1 21.770} C_DIS
LIN {X 0.050,Y -208.207,Z 284.099,A 0.000,B 0.000,C 90.000,E1 17.819} C_DIS
LIN {X -0.090,Y -203.114,Z 284.077,A 0.000,B 0.000,C 90.000,E1 13.883} C_DIS
LIN {X -0.029,Y -199.071,Z 284.055,A 0.000,B 0.000,C 90.000,E1 9.849} C_DIS
LIN {X -0.057,Y -195.536,Z 284.028,A 0.000,B 0.000,C 90.000,E1 4.992} C_DIS
LIN {X -0.094,Y -193.001,Z 283.993,A 0.000,B 0.000,C 90.000,E1 358.740} C_DIS
LIN {X -0.003,Y -194.400,Z 283.929,A 0.000,B 0.000,C 90.000,E1 347.229} C_DIS
LIN {X 0.076,Y -197.402,Z 283.902,A 0.000,B 0.000,C 90.000,E1 342.308} C_DIS
LIN {X -0.029,Y -201.121,Z 283.879,A 0.000,B 0.000,C 90.000,E1 338.284} C_DIS
LIN {X -0.089,Y -205.857,Z 283.857,A 0.000,B 0.000,C 90.000,E1 334.280} C_DIS
LIN {X 0.089,Y -211.583,Z 283.835,A 0.000,B 0.000,C 90.000,E1 330.255} C_DIS
LIN {X 0.053,Y -216.962,Z 283.817,A 0.000,B 0.000,C 90.000,E1 327.120} C_DIS
LIN {X -0.040,Y -223.130,Z 283.800,A 0.000,B 0.000,C 90.000,E1 324.036} C_DIS
LIN {X -0.028,Y -230.256,Z 283.783,A 0.000,B 0.000,C 90.000,E1 320.964} C_DIS
LIN {X 0.046,Y -239.306,Z 283.764,A 0.000,B 0.000,C 90.000,E1 317.553} C_DIS
LIN {X -0.144,Y -249.364,Z 283.746,A 0.000,B 0.000,C 90.000,E1 314.271} C_DIS
LIN {X -0.029,Y -260.478,Z 283.728,A 0.000,B 0.000,C 90.000,E1 310.987} C_DIS
LIN {X -0.076,Y -272.670,Z 283.710,A 0.000,B 0.000,C 90.000,E1 307.810} C_DIS
LIN {X 0.000,Y -284.705,Z 283.695,A 0.000,B 0.000,C 90.000,E1 305.025} C_DIS
LIN {X -0.099,Y -296.406,Z 283.681,A 0.000,B 0.000,C 90.000,E1 302.673} C_DIS
LIN {X 0.076,Y -313.090,Z 283.665,A 0.000,B 0.000,C 90.000,E1 299.667} C_DIS
LIN {X -0.036,Y -333.474,Z 283.647,A 0.000,B 0.000,C 90.000,E1 296.488} C_DIS
LIN {X -0.150,Y -348.443,Z 283.635,A 0.000,B 0.000,C 90.000,E1 294.335} C_DIS
LIN {X -0.094,Y -363.427,Z 283.623,A 0.000,B 0.000,C 90.000,E1 292.206} C_DIS
LIN {X -0.083,Y -376.517,Z 283.613,A 0.000,B 0.000,C 90.000,E1 290.429} C_DIS
LIN {X -0.140,Y -394.375,Z 283.601,A 0.000,B 0.000,C 90.000,E1 288.127} C_DIS
LIN {X 0.130,Y -405.567,Z 283.593,A 0.000,B 0.000,C 90.000,E1 286.677} C_DIS
LIN {X -0.096,Y -421.181,Z 283.582,A 0.000,B 0.000,C 90.000,E1 284.773} C_DIS
LIN {X 0.040,Y -427.755,Z 283.577,A 0.000,B 0.000,C 90.000,E1 283.939} C_DIS
LIN {X 0.127,Y -433.847,Z 283.573,A 0.000,B 0.000,C 90.000,E1 283.119} C_DIS
LIN {X -0.146,Y -439.509,Z 283.569,A 0.000,B 0.000,C 90.000,E1 282.355} C_DIS
LIN {X -0.158,Y -446.579,Z 283.563,A 0.000,B 0.000,C 90.000,E1 281.299} C_DIS
LIN {X -0.171,Y -453.163,Z 283.557,A 0.000,B 0.000,C 90.000,E1 280.254} C_DIS
LIN {X 0.169,Y -460.829,Z 283.550,A 0.000,B 0.000,C 90.000,E1 278.916} C_DIS
LIN {X -0.197,Y -466.541,Z 283.544,A 0.000,B 0.000,C 90.000,E1 277.936} C_DIS
LIN {X -0.184,Y -473.257,Z 283.537,A 0.000,B 0.000,C 90.000,E1 276.663} C_DIS
LIN {X -0.219,Y -476.958,Z 283.533,A 0.000,B 0.000,C 90.000,E1 275.910} C_DIS
LIN {X -0.084,Y -479.147,Z 283.530,A 0.000,B 0.000,C 90.000,E1 275.391} C_DIS
LIN {X 0.023,Y -481.050,Z 283.527,A 0.000,B 0.000,C 90.000,E1 274.878} C_DIS
LIN {X 0.181,Y -482.574,Z 283.524,A 0.000,B 0.000,C 90.000,E1 274.359} C_DIS
LIN {X -0.135,Y -483.680,Z 283.522,A 0.000,B 0.000,C 90.000,E1 273.898} C_DIS
LIN {X 0.008,Y -484.437,Z 283.519,A 0.000,B 0.000,C 90.000,E1 273.383} C_DIS
LIN {X 0.186,Y -484.825,Z 283.516,A 0.000,B 0.000,C 90.000,E1 272.865} C_DIS
LIN {X 0.022,Y -484.770,Z 283.511,A 0.000,B 0.000,C 90.000,E1 271.892} C_DIS
LIN {X -0.122,Y -484.135,Z 283.505,A 0.000,B 0.000,C 90.000,E1 270.917} C_DIS
LIN {X 0.040,Y -483.561,Z 283.502,A 0.000,B 0.000,C 90.000,E1 270.401} C_DIS
LIN {X 0.200,Y -482.680,Z 283.499,A 0.000,B 0.000,C 90.000,E1 269.885} C_DIS
LIN {X -0.126,Y -481.327,Z 283.497,A 0.000,B 0.000,C 90.000,E1 269.427} C_DIS
LIN {X 0.024,Y -479.476,Z 283.494,A 0.000,B 0.000,C 90.000,E1 268.912} C_DIS
LIN {X 0.165,Y -476.963,Z 283.491,A 0.000,B 0.000,C 90.000,E1 268.396} C_DIS
LIN {X -0.172,Y -473.660,Z 283.488,A 0.000,B 0.000,C 90.000,E1 267.936} C_DIS
LIN {X -0.067,Y -469.392,Z 283.486,A 0.000,B 0.000,C 90.000,E1 267.421} C_DIS
LIN {X 0.206,Y -466.915,Z 283.484,A 0.000,B 0.000,C 90.000,E1 267.135} C_DIS
LIN {X 0.024,Y -461.185,Z 283.482,A 0.000,B 0.000,C 90.000,E1 266.674} C_DIS
LIN {X 0.011,Y -457.880,Z 283.480,A 0.000,B 0.000,C 90.000,E1 266.445} C_DIS
LIN {X -0.172,Y -454.697,Z 283.479,A 0.000,B 0.000,C 90.000,E1 266.274} C_DIS
LIN {X 0.096,Y -450.949,Z 283.478,A 0.000,B 0.000,C 90.000,E1 266.045} C_DIS
LIN {X -0.182,Y -447.470,Z 283.477,A 0.000,B 0.000,C 90.000,E1 265.927} C_DIS
LIN {X -0.016,Y -439.579,Z 283.476,A 0.000,B 0.000,C 90.000,E1 265.641} C_DIS
LIN {X -0.098,Y -430.570,Z 283.475,A 0.000,B 0.000,C 90.000,E1 265.469} C_DIS
LIN {X -0.201,Y -424.935,Z 283.474,A 0.000,B 0.000,C 90.000,E1 265.412} C_DIS
LIN {X -0.105,Y -419.007,Z 283.474,A 0.000,B 0.000,C 90.000,E1 265.355} C_DIS
LIN {X -0.081,Y -180.905,Z 283.474,A 0.000,B 0.000,C 90.000,E1 265.355} C_DIS
LIN {X -0.056,Y -180.243,Z 283.465,A 0.000,B 0.000,C 90.000,E1 263.628} C_DIS
LIN {X -0.037,Y -178.730,Z 283.441,A 0.000,B 0.000,C 90.000,E1 259.398} C_DIS
LIN {X 0.031,Y -175.778,Z 283.413,A 0.000,B 0.000,C 90.000,E1 254.283} C_DIS
LIN {X 0.018,Y -171.961,Z 283.384,A 0.000,B 0.000,C 90.000,E1 249.156} C_DIS
LIN {X 0.056,Y -171.357,Z 283.379,A 0.000,B 0.000,C 90.000,E1 248.284} C_DIS
LIN {X 0.033,Y -167.606,Z 283.355,A 0.000,B 0.000,C 90.000,E1 243.973} C_DIS
LIN {X 0.046,Y -166.252,Z 283.346,A 0.000,B 0.000,C 90.000,E1 242.231} C_DIS
LIN {X 0.033,Y -163.008,Z 283.326,A 0.000,B 0.000,C 90.000,E1 238.742} C_DIS
LIN {X 0.079,Y -160.929,Z 283.312,A 0.000,B 0.000,C 90.000,E1 236.087} C_DIS
LIN {X 0.056,Y -157.690,Z 283.292,A 0.000,B 0.000,C 90.000,E1 232.557} C_DIS
LIN {X -0.005,Y -155.730,Z 283.277,A 0.000,B 0.000,C 90.000,E1 229.908} C_DIS
LIN {X 0.048,Y -151.988,Z 283.252,A 0.000,B 0.000,C 90.000,E1 225.405} C_DIS
LIN {X 0.064,Y -150.233,Z 283.237,A 0.000,B 0.000,C 90.000,E1 222.690} C_DIS
LIN {X -0.013,Y -146.994,Z 283.212,A 0.000,B 0.000,C 90.000,E1 218.177} C_DIS
LIN {X -0.023,Y -145.579,Z 283.197,A 0.000,B 0.000,C 90.000,E1 215.438} C_DIS
LIN {X -0.028,Y -142.968,Z 283.171,A 0.000,B 0.000,C 90.000,E1 210.846} C_DIS
LIN {X 0.025,Y -141.594,Z 283.151,A 0.000,B 0.000,C 90.000,E1 207.129} C_DIS
LIN {X 0.071,Y -139.421,Z 283.115,A 0.000,B 0.000,C 90.000,E1 200.610} C_DIS
LIN {X -0.008,Y -139.148,Z 283.104,A 0.000,B 0.000,C 90.000,E1 198.779} C_DIS
LIN {X 0.014,Y -138.346,Z 283.058,A 0.000,B 0.000,C 90.000,E1 190.366} C_DIS
LIN {X 0.000,Y -139.488,Z 283.006,A 0.000,B 0.000,C 90.000,E1 181.031} C_DIS
LIN {X -0.061,Y -141.090,Z 282.975,A 0.000,B 0.000,C 90.000,E1 175.469} C_DIS
LIN {X 0.034,Y -142.467,Z 282.959,A 0.000,B 0.000,C 90.000,E1 172.648} C_DIS
LIN {X -0.018,Y -144.712,Z 282.934,A 0.000,B 0.000,C 90.000,E1 168.049} C_DIS
LIN {X -0.066,Y -147.311,Z 282.913,A 0.000,B 0.000,C 90.000,E1 164.393} C_DIS
LIN {X -0.051,Y -150.632,Z 282.888,A 0.000,B 0.000,C 90.000,E1 159.826} C_DIS
LIN {X 0.024,Y -154.109,Z 282.868,A 0.000,B 0.000,C 90.000,E1 156.177} C_DIS
LIN {X -0.052,Y -157.533,Z 282.848,A 0.000,B 0.000,C 90.000,E1 152.615} C_DIS
LIN {X -0.108,Y -161.770,Z 282.828,A 0.000,B 0.000,C 90.000,E1 149.076} C_DIS
LIN {X -0.003,Y -165.962,Z 282.808,A 0.000,B 0.000,C 90.000,E1 145.515} C_DIS
LIN {X -0.006,Y -170.955,Z 282.789,A 0.000,B 0.000,C 90.000,E1 142.029} C_DIS
LIN {X 0.046,Y -175.824,Z 282.770,A 0.000,B 0.000,C 90.000,E1 138.566} C_DIS
LIN {X 0.040,Y -181.431,Z 282.751,A 0.000,B 0.000,C 90.000,E1 135.162} C_DIS
LIN {X -0.085,Y -186.936,Z 282.732,A 0.000,B 0.000,C 90.000,E1 131.838} C_DIS
LIN {X -0.013,Y -191.513,Z 282.718,A 0.000,B 0.000,C 90.000,E1 129.322} C_DIS
LIN {X 0.072,Y -197.380,Z 282.700,A 0.000,B 0.000,C 90.000,E1 126.011} C_DIS
LIN {X -0.004,Y -200.655,Z 282.691,A 0.000,B 0.000,C 90.000,E1 124.405} C_DIS
LIN {X 0.058,Y -203.010,Z 282.684,A 0.000,B 0.000,C 90.000,E1 123.038} C_DIS
LIN {X 0.041,Y -305.548,Z 282.684,A 0.000,B 0.000,C 90.000,E1 123.038} C_DIS
LIN {X -0.054,Y -306.583,Z 282.684,A 0.000,B 0.000,C 90.000,E1 123.038} C_DIS
LIN {X -0.065,Y -311.714,Z 282.682,A 0.000,B 0.000,C 90.000,E1 122.801} C_DIS
LIN {X 0.006,Y -314.872,Z 282.681,A 0.000,B 0.000,C 90.000,E1 122.498} C_DIS
LIN {X -0.176,Y -318.529,Z 282.678,A 0.000,B 0.000,C 90.000,E1 122.005} C_DIS
LIN {X -0.110,Y -320.105,Z 282.676,A 0.000,B 0.000,C 90.000,E1 121.671} C_DIS
LIN {X 0.059,Y -333.898,Z 282.656,A 0.000,B 0.000,C 90.000,E1 118.153} C_DIS
LIN {X -0.079,Y -346.698,Z 282.641,A 0.000,B 0.000,C 90.000,E1 115.387} C_DIS
LIN {X -0.031,Y -359.378,Z 282.627,A 0.000,B 0.000,C 90.000,E1 112.950} C_DIS
LIN {X 0.078,Y -373.380,Z 282.614,A 0.000,B 0.000,C 90.000,E1 110.556} C_DIS
LIN {X 0.060,Y -388.806,Z 282.601,A 0.000,B 0.000,C 90.000,E1 108.236} C_DIS
LIN {X 0.063,Y -405.771,Z 282.589,A 0.000,B 0.000,C 90.000,E1 105.969} C_DIS
LIN {X -0.012,Y -424.401,Z 282.577,A 0.000,B 0.000,C 90.000,E1 103.772} C_DIS
LIN {X 0.089,Y -444.382,Z 282.565,A 0.000,B 0.000,C 90.000,E1 101.658} C_DIS
LIN {X 0.141,Y -464.953,Z 282.554,A 0.000,B 0.000,C 90.000,E1 99.726} C_DIS
LIN {X 0.062,Y -488.699,Z 282.543,A 0.000,B 0.000,C 90.000,E1 97.757} C_DIS
LIN {X -0.024,Y -499.422,Z 282.539,A 0.000,B 0.000,C 90.000,E1 96.947} C_DIS
LIN {X -0.058,Y -503.423,Z 282.536,A 0.000,B 0.000,C 90.000,E1 96.549} C_DIS
LIN {X -0.122,Y -505.019,Z 282.535,A 0.000,B 0.000,C 90.000,E1 96.315} C_DIS
LIN {X -0.242,Y -506.214,Z 282.534,A 0.000,B 0.000,C 90.000,E1 96.087} C_DIS
LIN {X 0.076,Y -507.663,Z 282.531,A 0.000,B 0.000,C 90.000,E1 95.568} C_DIS
LIN {X -0.105,Y -508.046,Z 282.528,A 0.000,B 0.000,C 90.000,E1 95.106} C_DIS
LIN {X 0.225,Y -507.421,Z 282.526,A 0.000,B 0.000,C 90.000,E1 94.588} C_DIS
LIN {X 0.014,Y -505.677,Z 282.523,A 0.000,B 0.000,C 90.000,E1 94.131} C_DIS
LIN {X -0.058,Y -504.282,Z 282.522,A 0.000,B 0.000,C 90.000,E1 93.898} C_DIS
LIN {X 0.015,Y -496.829,Z 282.516,A 0.000,B 0.000,C 90.000,E1 92.922} C_DIS
LIN {X -0.013,Y -488.627,Z 282.511,A 0.000,B 0.000,C 90.000,E1 91.949} C_DIS
LIN {X 0.059,Y -465.591,Z 282.496,A 0.000,B 0.000,C 90.000,E1 89.198} C_DIS
LIN {X -0.050,Y -452.269,Z 282.486,A 0.000,B 0.000,C 90.000,E1 87.421} C_DIS
LIN {X -0.087,Y -433.220,Z 282.470,A 0.000,B 0.000,C 90.000,E1 84.546} C_DIS
LIN {X 0.080,Y -417.522,Z 282.455,A 0.000,B 0.000,C 90.000,E1 81.837} C_DIS
LIN {X -0.033,Y -403.271,Z 282.439,A 0.000,B 0.000,C 90.000,E1 79.106} C_DIS
LIN {X 0.173,Y -393.202,Z 282.429,A 0.000,B 0.000,C 90.000,E1 77.117} C_DIS
LIN {X -0.124,Y -383.195,Z 282.418,A 0.000,B 0.000,C 90.000,E1 75.172} C_DIS
LIN {X -0.058,Y -373.251,Z 282.406,A 0.000,B 0.000,C 90.000,E1 73.142} C_DIS
LIN {X -0.010,Y -361.844,Z 282.393,A 0.000,B 0.000,C 90.000,E1 70.786} C_DIS
LIN {X -0.077,Y -349.341,Z 282.378,A 0.000,B 0.000,C 90.000,E1 68.103} C_DIS
LIN {X 0.022,Y -333.913,Z 282.358,A 0.000,B 0.000,C 90.000,E1 64.409} C_DIS
LIN {X -0.085,Y -321.174,Z 282.339,A 0.000,B 0.000,C 90.000,E1 60.973} C_DIS
LIN {X 0.014,Y -311.196,Z 282.323,A 0.000,B 0.000,C 90.000,E1 58.074} C_DIS
LIN {X 0.027,Y -300.706,Z 282.305,A 0.000,B 0.000,C 90.000,E1 54.815} C_DIS
LIN {X -0.093,Y -292.482,Z 282.290,A 0.000,B 0.000,C 90.000,E1 52.190} C_DIS
LIN {X 0.046,Y -286.335,Z 282.279,A 0.000,B 0.000,C 90.000,E1 50.150} C_DIS
LIN {X -0.153,Y -278.072,Z 282.264,A 0.000,B 0.000,C 90.000,E1 47.472} C_DIS
LIN {X 0.168,Y -268.353,Z 282.244,A 0.000,B 0.000,C 90.000,E1 43.947} C_DIS
LIN {X 0.100,Y -260.931,Z 282.229,A 0.000,B 0.000,C 90.000,E1 41.148} C_DIS
LIN {X -0.005,Y -255.330,Z 282.217,A 0.000,B 0.000,C 90.000,E1 39.036} C_DIS
LIN {X 0.021,Y -249.615,Z 282.205,A 0.000,B 0.000,C 90.000,E1 36.870} C_DIS
LIN {X -0.002,Y -243.711,Z 282.193,A 0.000,B 0.000,C 90.000,E1 34.692} C_DIS
LIN {X -0.040,Y -233.957,Z 282.172,A 0.000,B 0.000,C 90.000,E1 31.003} C_DIS
LIN {X 0.030,Y -226.800,Z 282.155,A 0.000,B 0.000,C 90.000,E1 27.975} C_DIS
LIN {X 0.108,Y -220.362,Z 282.138,A 0.000,B 0.000,C 90.000,E1 24.899} C_DIS
LIN {X -0.048,Y -214.698,Z 282.121,A 0.000,B 0.000,C 90.000,E1 21.844} C_DIS
LIN {X -0.066,Y -208.570,Z 282.099,A 0.000,B 0.000,C 90.000,E1 17.928} C_DIS
LIN {X -0.004,Y -203.439,Z 282.077,A 0.000,B 0.000,C 90.000,E1 13.939} C_DIS
LIN {X 0.063,Y -199.379,Z 282.055,A 0.000,B 0.000,C 90.000,E1 9.905} C_DIS
LIN {X 0.041,Y -195.817,Z 282.028,A 0.000,B 0.000,C 90.000,E1 5.049} C_DIS
LIN {X -0.093,Y -193.209,Z 281.993,A 0.000,B 0.000,C 90.000,E1 358.740} C_DIS
LIN {X 0.016,Y -194.580,Z 281.929,A 0.000,B 0.000,C 90.000,E1 347.229} C_DIS
LIN {X -0.086,Y -197.576,Z 281.902,A 0.000,B 0.000,C 90.000,E1 342.362} C_DIS
LIN {X 0.003,Y -201.287,Z 281.879,A 0.000,B 0.000,C 90.000,E1 338.284} C_DIS
LIN {X -0.051,Y -206.003,Z 281.857,A 0.000,B 0.000,C 90.000,E1 334.280} C_DIS
LIN {X 0.028,Y -211.734,Z 281.835,A 0.000,B 0.000,C 90.000,E1 330.284} C_DIS
LIN {X -0.081,Y -217.141,Z 281.817,A 0.000,B 0.000,C 90.000,E1 327.168} C_DIS
LIN {X 0.013,Y -223.333,Z 281.800,A 0.000,B 0.000,C 90.000,E1 324.036} C_DIS
LIN {X 0.033,Y -230.482,Z 281.783,A 0.000,B 0.000,C 90.000,E1 320.964} C_DIS
LIN {X 0.116,Y -239.518,Z 281.764,A 0.000,B 0.000,C 90.000,E1 317.553} C_DIS
LIN {X -0.065,Y -249.575,Z 281.746,A 0.000,B 0.000,C 90.000,E1 314.271} C_DIS
LIN {X 0.060,Y -260.674,Z 281.728,A 0.000,B 0.000,C 90.000,E1 310.987} C_DIS
LIN {X 0.023,Y -272.863,Z 281.710,A 0.000,B 0.000,C 90.000,E1 307.810} C_DIS
LIN {X 0.108,Y -284.904,Z 281.695,A 0.000,B 0.000,C 90.000,E1 305.025} C_DIS
LIN {X 0.013,Y -298.400,Z 281.680,A 0.000,B 0.000,C 90.000,E1 302.339} C_DIS
LIN {X -0.168,Y -315.245,Z 281.663,A 0.000,B 0.000,C 90.000,E1 299.411} C_DIS
LIN {X 0.079,Y -335.808,Z 281.646,A 0.000,B 0.000,C 90.000,E1 296.181} C_DIS
LIN {X 0.006,Y -348.614,Z 281.635,A 0.000,B 0.000,C 90.000,E1 294.335} C_DIS
LIN {X 0.020,Y -361.403,Z 281.625,A 0.000,B 0.000,C 90.000,E1 292.514} C_DIS
LIN {X 0.092,Y -376.603,Z 281.614,A 0.000,B 0.000,C 90.000,E1 290.429} C_DIS
LIN {X 0.015,Y -392.141,Z 281.602,A 0.000,B 0.000,C 90.000,E1 288.417} C_DIS
LIN {X -0.067,Y -405.539,Z 281.593,A 0.000,B 0.000,C 90.000,E1 286.732} C_DIS
LIN {X 0.102,Y -421.100,Z 281.582,A 0.000,B 0.000,C 90.000,E1 284.773} C_DIS
LIN {X -0.019,Y -429.728,Z 281.576,A 0.000,B 0.000,C 90.000,E1 283.703} C_DIS
LIN {X -0.143,Y -437.541,Z 281.570,A 0.000,B 0.000,C 90.000,E1 282.647} C_DIS
LIN {X -0.177,Y -444.709,Z 281.564,A 0.000,B 0.000,C 90.000,E1 281.591} C_DIS
LIN {X -0.215,Y -451.391,Z 281.558,A 0.000,B 0.000,C 90.000,E1 280.546} C_DIS
LIN {X 0.103,Y -459.150,Z 281.551,A 0.000,B 0.000,C 90.000,E1 279.208} C_DIS
LIN {X -0.215,Y -464.939,Z 281.546,A 0.000,B 0.000,C 90.000,E1 278.219} C_DIS
LIN {X 0.233,Y -471.745,Z 281.538,A 0.000,B 0.000,C 90.000,E1 276.891} C_DIS
LIN {X -0.013,Y -476.749,Z 281.533,A 0.000,B 0.000,C 90.000,E1 275.910} C_DIS
LIN {X 0.123,Y -478.946,Z 281.530,A 0.000,B 0.000,C 90.000,E1 275.391} C_DIS
LIN {X -0.249,Y -480.851,Z 281.527,A 0.000,B 0.000,C 90.000,E1 274.935} C_DIS
LIN {X -0.094,Y -482.386,Z 281.524,A 0.000,B 0.000,C 90.000,E1 274.416} C_DIS
LIN {X 0.070,Y -483.524,Z 281.522,A 0.000,B 0.000,C 90.000,E1 273.898} C_DIS
LIN {X 0.212,Y -484.276,Z 281.519,A 0.000,B 0.000,C 90.000,E1 273.383} C_DIS
LIN {X -0.095,Y -484.688,Z 281.516,A 0.000,B 0.000,C 90.000,E1 272.922} C_DIS
LIN {X 0.062,Y -484.779,Z 281.513,A 0.000,B 0.000,C 90.000,E1 272.407} C_DIS
LIN {X -0.083,Y -484.449,Z 281.508,A 0.000,B 0.000,C 90.000,E1 271.432} C_DIS
LIN {X 0.078,Y -484.112,Z 281.505,A 0.000,B 0.000,C 90.000,E1 270.917} C_DIS
LIN {X 0.240,Y -483.557,Z 281.502,A 0.000,B 0.000,C 90.000,E1 270.401} C_DIS
LIN {X -0.083,Y -482.681,Z 281.500,A 0.000,B 0.000,C 90.000,E1 269.943} C_DIS
LIN {X 0.073,Y -481.368,Z 281.497,A 0.000,B 0.000,C 90.000,E1 269.427} C_DIS
LIN {X 0.224,Y -479.532,Z 281.494,A 0.000,B 0.000,C 90.000,E1 268.912} C_DIS
LIN {X -0.114,Y -477.050,Z 281.491,A 0.000,B 0.000,C 90.000,E1 268.453} C_DIS
LIN {X 0.024,Y -473.825,Z 281.489,A 0.000,B 0.000,C 90.000,E1 267.936} C_DIS
LIN {X 0.129,Y -469.672,Z 281.486,A 0.000,B 0.000,C 90.000,E1 267.421} C_DIS
LIN {X -0.065,Y -467.220,Z 281.484,A 0.000,B 0.000,C 90.000,E1 267.192} C_DIS
LIN {X 0.187,Y -461.583,Z 281.482,A 0.000,B 0.000,C 90.000,E1 266.674} C_DIS
LIN {X 0.140,Y -458.274,Z 281.480,A 0.000,B 0.000,C 90.000,E1 266.445} C_DIS
LIN {X -0.063,Y -455.121,Z 281.479,A 0.000,B 0.000,C 90.000,E1 266.274} C_DIS
LIN {X 0.186,Y -451.474,Z 281.478,A 0.000,B 0.000,C 90.000,E1 266.045} C_DIS
LIN {X -0.132,Y -447.991,Z 281.477,A 0.000,B 0.000,C 90.000,E1 265.927} C_DIS
LIN {X -0.031,Y -440.108,Z 281.476,A 0.000,B 0.000,C 90.000,E1 265.641} C_DIS
LIN {X -0.153,Y -431.074,Z 281.475,A 0.000,B 0.000,C 90.000,E1 265.469} C_DIS
LIN {X 0.150,Y -425.712,Z 281.474,A 0.000,B 0.000,C 90.000,E1 265.355} C_DIS
LIN {X -0.197,Y -420.228,Z 281.474,A 0.000,B 0.000,C 90.000,E1 265.355} C_DIS
LIN {X 0.134,Y -414.868,Z 281.474,A 0.000,B 0.000,C 90.000,E1 265.298} C_DIS
LIN {X 0.040,Y -180.905,Z 281.474,A 0.000,B 0.000,C 90.000,E1 265.298} C_DIS
LIN {X 0.076,Y -180.236,Z 281.464,A 0.000,B 0.000,C 90.000,E1 263.571} C_DIS
LIN {X -0.083,Y -178.720,Z 281.441,A 0.000,B 0.000,C 90.000,E1 259.398} C_DIS
LIN {X -0.015,Y -175.769,Z 281.413,A 0.000,B 0.000,C 90.000,E1 254.283} C_DIS
LIN {X 0.034,Y -171.953,Z 281.384,A 0.000,B 0.000,C 90.000,E1 249.135} C_DIS
LIN {X 0.010,Y -171.343,Z 281.379,A 0.000,B 0.000,C 90.000,E1 248.284} C_DIS
LIN {X -0.012,Y -167.596,Z 281.355,A 0.000,B 0.000,C 90.000,E1 243.973} C_DIS
LIN {X 0.000,Y -166.236,Z 281.346,A 0.000,B 0.000,C 90.000,E1 242.231} C_DIS
LIN {X -0.011,Y -162.995,Z 281.326,A 0.000,B 0.000,C 90.000,E1 238.742} C_DIS
LIN {X 0.036,Y -160.914,Z 281.312,A 0.000,B 0.000,C 90.000,E1 236.087} C_DIS
LIN {X 0.013,Y -157.678,Z 281.292,A 0.000,B 0.000,C 90.000,E1 232.557} C_DIS
LIN {X -0.048,Y -155.716,Z 281.277,A 0.000,B 0.000,C 90.000,E1 229.908} C_DIS
LIN {X 0.006,Y -151.977,Z 281.252,A 0.000,B 0.000,C 90.000,E1 225.405} C_DIS
LIN {X 0.022,Y -150.220,Z 281.237,A 0.000,B 0.000,C 90.000,E1 222.690} C_DIS
LIN {X -0.054,Y -146.984,Z 281.212,A 0.000,B 0.000,C 90.000,E1 218.177} C_DIS
LIN {X 0.054,Y -145.570,Z 281.197,A 0.000,B 0.000,C 90.000,E1 215.391} C_DIS
LIN {X 0.054,Y -142.960,Z 281.171,A 0.000,B 0.000,C 90.000,E1 210.797} C_DIS
LIN {X -0.015,Y -141.587,Z 281.151,A 0.000,B 0.000,C 90.000,E1 207.129} C_DIS
LIN {X 0.031,Y -139.418,Z 281.115,A 0.000,B 0.000,C 90.000,E1 200.610} C_DIS
LIN {X -0.048,Y -139.144,Z 281.104,A 0.000,B 0.000,C 90.000,E1 198.779} C_DIS
LIN {X -0.026,Y -138.347,Z 281.058,A 0.000,B 0.000,C 90.000,E1 190.366} C_DIS
LIN {X -0.040,Y -139.490,Z 281.006,A 0.000,B 0.000,C 90.000,E1 181.031} C_DIS
LIN {X 0.040,Y -141.097,Z 280.975,A 0.000,B 0.000,C 90.000,E1 175.412} C_DIS
LIN {X -0.006,Y -142.475,Z 280.959,A 0.000,B 0.000,C 90.000,E1 172.648} C_DIS
LIN {X -0.059,Y -144.722,Z 280.933,A 0.000,B 0.000,C 90.000,E1 168.049} C_DIS
LIN {X 0.033,Y -147.324,Z 280.913,A 0.000,B 0.000,C 90.000,E1 164.338} C_DIS
LIN {X -0.042,Y -150.647,Z 280.888,A 0.000,B 0.000,C 90.000,E1 159.806} C_DIS
LIN {X -0.019,Y -154.124,Z 280.868,A 0.000,B 0.000,C 90.000,E1 156.177} C_DIS
LIN {X 0.044,Y -157.550,Z 280.848,A 0.000,B 0.000,C 90.000,E1 152.564} C_DIS
LIN {X 0.070,Y -161.791,Z 280.828,A 0.000,B 0.000,C 90.000,E1 148.997} C_DIS
LIN {X -0.048,Y -165.982,Z 280.808,A 0.000,B 0.000,C 90.000,E1 145.515} C_DIS
LIN {X -0.052,Y -170.979,Z 280.789,A 0.000,B 0.000,C 90.000,E1 142.029} C_DIS
LIN {X -0.001,Y -175.848,Z 280.770,A 0.000,B 0.000,C 90.000,E1 138.566} C_DIS
LIN {X -0.007,Y -181.453,Z 280.751,A 0.000,B 0.000,C 90.000,E1 135.162} C_DIS
LIN {X 0.131,Y -186.963,Z 280.732,A 0.000,B 0.000,C 90.000,E1 131.757} C_DIS
LIN {X -0.013,Y -190.077,Z 280.723,A 0.000,B 0.000,C 90.000,E1 130.135} C_DIS
LIN {X -0.121,Y -195.850,Z 280.705,A 0.000,B 0.000,C 90.000,E1 126.870} C_DIS
LIN {X -0.054,Y -200.681,Z 280.691,A 0.000,B 0.000,C 90.000,E1 124.405} C_DIS
LIN {X 0.021,Y -203.086,Z 280.683,A 0.000,B 0.000,C 90.000,E1 123.007} C_DIS
LIN {X -0.010,Y -305.174,Z 280.683,A 0.000,B 0.000,C 90.000,E1 123.007} C_DIS
LIN {X 0.123,Y -306.737,Z 280.683,A 0.000,B 0.000,C 90.000,E1 122.959} C_DIS
LIN {X 0.119,Y -311.405,Z 280.682,A 0.000,B 0.000,C 90.000,E1 122.752} C_DIS
LIN {X -0.001,Y -314.605,Z 280.681,A 0.000,B 0.000,C 90.000,E1 122.498} C_DIS
LIN {X -0.048,Y -318.282,Z 280.678,A 0.000,B 0.000,C 90.000,E1 122.005} C_DIS
LIN {X 0.017,Y -319.945,Z 280.676,A 0.000,B 0.000,C 90.000,E1 121.671} C_DIS
LIN {X 0.071,Y -332.450,Z 280.658,A 0.000,B 0.000,C 90.000,E1 118.487} C_DIS
LIN {X -0.104,Y -345.076,Z 280.643,A 0.000,B 0.000,C 90.000,E1 115.720} C_DIS
LIN {X 0.051,Y -357.587,Z 280.629,A 0.000,B 0.000,C 90.000,E1 113.259} C_DIS
LIN {X 0.114,Y -371.406,Z 280.616,A 0.000,B 0.000,C 90.000,E1 110.865} C_DIS
LIN {X 0.052,Y -386.636,Z 280.603,A 0.000,B 0.000,C 90.000,E1 108.544} C_DIS
LIN {X 0.117,Y -403.388,Z 280.590,A 0.000,B 0.000,C 90.000,E1 106.260} C_DIS
LIN {X -0.020,Y -421.788,Z 280.578,A 0.000,B 0.000,C 90.000,E1 104.064} C_DIS
LIN {X -0.094,Y -441.662,Z 280.566,A 0.000,B 0.000,C 90.000,E1 101.951} C_DIS
LIN {X 0.226,Y -462.161,Z 280.556,A 0.000,B 0.000,C 90.000,E1 99.962} C_DIS
LIN {X -0.016,Y -485.811,Z 280.544,A 0.000,B 0.000,C 90.000,E1 97.992} C_DIS
LIN {X 0.092,Y -499.214,Z 280.539,A 0.000,B 0.000,C 90.000,E1 96.947} C_DIS
LIN {X 0.098,Y -503.369,Z 280.536,A 0.000,B 0.000,C 90.000,E1 96.549} C_DIS
LIN {X 0.094,Y -504.997,Z 280.535,A 0.000,B 0.000,C 90.000,E1 96.315} C_DIS
LIN {X 0.034,Y -506.228,Z 280.534,A 0.000,B 0.000,C 90.000,E1 96.087} C_DIS
LIN {X -0.153,Y -507.793,Z 280.531,A 0.000,B 0.000,C 90.000,E1 95.625} C_DIS
LIN {X 0.172,Y -508.275,Z 280.528,A 0.000,B 0.000,C 90.000,E1 95.106} C_DIS
LIN {X -0.003,Y -507.752,Z 280.526,A 0.000,B 0.000,C 90.000,E1 94.645} C_DIS
LIN {X -0.214,Y -506.132,Z 280.523,A 0.000,B 0.000,C 90.000,E1 94.188} C_DIS
LIN {X 0.220,Y -504.817,Z 280.522,A 0.000,B 0.000,C 90.000,E1 93.898} C_DIS
LIN {X -0.109,Y -499.405,Z 280.518,A 0.000,B 0.000,C 90.000,E1 93.212} C_DIS
LIN {X -0.084,Y -491.371,Z 280.512,A 0.000,B 0.000,C 90.000,E1 92.236} C_DIS
LIN {X 0.011,Y -478.557,Z 280.504,A 0.000,B 0.000,C 90.000,E1 90.745} C_DIS
LIN {X 0.195,Y -460.277,Z 280.492,A 0.000,B 0.000,C 90.000,E1 88.453} C_DIS
LIN {X -0.046,Y -443.917,Z 280.479,A 0.000,B 0.000,C 90.000,E1 86.159} C_DIS
LIN {X 0.118,Y -425.674,Z 280.462,A 0.000,B 0.000,C 90.000,E1 83.223} C_DIS
LIN {X 0.047,Y -412.190,Z 280.449,A 0.000,B 0.000,C 90.000,E1 80.792} C_DIS
LIN {X -0.027,Y -402.332,Z 280.438,A 0.000,B 0.000,C 90.000,E1 78.870} C_DIS
LIN {X -0.156,Y -390.850,Z 280.426,A 0.000,B 0.000,C 90.000,E1 76.645} C_DIS
LIN {X 0.123,Y -378.042,Z 280.411,A 0.000,B 0.000,C 90.000,E1 74.031} C_DIS
LIN {X 0.078,Y -368.058,Z 280.400,A 0.000,B 0.000,C 90.000,E1 72.000} C_DIS
LIN {X -0.007,Y -356.766,Z 280.387,A 0.000,B 0.000,C 90.000,E1 69.645} C_DIS
LIN {X 0.079,Y -340.703,Z 280.367,A 0.000,B 0.000,C 90.000,E1 65.997} C_DIS
LIN {X -0.008,Y -326.190,Z 280.346,A 0.000,B 0.000,C 90.000,E1 62.281} C_DIS
LIN {X -0.004,Y -317.228,Z 280.332,A 0.000,B 0.000,C 90.000,E1 59.744} C_DIS
LIN {X 0.050,Y -307.441,Z 280.316,A 0.000,B 0.000,C 90.000,E1 56.834} C_DIS
LIN {X 0.162,Y -299.121,Z 280.301,A 0.000,B 0.000,C 90.000,E1 54.196} C_DIS
LIN {X 0.171,Y -290.900,Z 280.286,A 0.000,B 0.000,C 90.000,E1 51.537} C_DIS
LIN {X 0.054,Y -284.724,Z 280.275,A 0.000,B 0.000,C 90.000,E1 49.542} C_DIS
LIN {X 0.012,Y -274.528,Z 280.256,A 0.000,B 0.000,C 90.000,E1 46.134} C_DIS
LIN {X -0.104,Y -266.893,Z 280.241,A 0.000,B 0.000,C 90.000,E1 43.380} C_DIS
LIN {X 0.077,Y -261.342,Z 280.229,A 0.000,B 0.000,C 90.000,E1 41.229} C_DIS
LIN {X -0.020,Y -255.727,Z 280.217,A 0.000,B 0.000,C 90.000,E1 39.116} C_DIS
LIN {X 0.018,Y -250.030,Z 280.205,A 0.000,B 0.000,C 90.000,E1 36.950} C_DIS
LIN {X 0.003,Y -244.140,Z 280.193,A 0.000,B 0.000,C 90.000,E1 34.771} C_DIS
LIN {X -0.018,Y -234.411,Z 280.173,A 0.000,B 0.000,C 90.000,E1 31.082} C_DIS
LIN {X -0.132,Y -227.234,Z 280.156,A 0.000,B 0.000,C 90.000,E1 28.103} C_DIS
LIN {X -0.040,Y -220.783,Z 280.139,A 0.000,B 0.000,C 90.000,E1 25.027} C_DIS
LIN {X 0.100,Y -215.121,Z 280.122,A 0.000,B 0.000,C 90.000,E1 21.897} C_DIS
LIN {X 0.020,Y -208.963,Z 280.100,A 0.000,B 0.000,C 90.000,E1 18.000} C_DIS
LIN {X -0.096,Y -203.788,Z 280.078,A 0.000,B 0.000,C 90.000,E1 14.064} C_DIS
LIN {X 0.026,Y -199.707,Z 280.056,A 0.000,B 0.000,C 90.000,E1 10.018} C_DIS
LIN {X 0.012,Y -196.099,Z 280.029,A 0.000,B 0.000,C 90.000,E1 5.163} C_DIS
LIN {X -0.092,Y -193.413,Z 279.993,A 0.000,B 0.000,C 90.000,E1 358.740} C_DIS
LIN {X 0.035,Y -194.767,Z 279.929,A 0.000,B 0.000,C 90.000,E1 347.229} C_DIS
LIN {X -0.060,Y -197.756,Z 279.902,A 0.000,B 0.000,C 90.000,E1 342.362} C_DIS
LIN {X 0.034,Y -201.456,Z 279.879,A 0.000,B 0.000,C 90.000,E1 338.284} C_DIS
LIN {X -0.013,Y -206.156,Z 279.857,A 0.000,B 0.000,C 90.000,E1 334.280} C_DIS
LIN {X -0.113,Y -211.883,Z 279.835,A 0.000,B 0.000,C 90.000,E1 330.333} C_DIS
LIN {X -0.033,Y -217.323,Z 279.818,A 0.000,B 0.000,C 90.000,E1 327.168} C_DIS
LIN {X -0.062,Y -223.537,Z 279.800,A 0.000,B 0.000,C 90.000,E1 324.069} C_DIS
LIN {X -0.083,Y -230.717,Z 279.783,A 0.000,B 0.000,C 90.000,E1 321.009} C_DIS
LIN {X 0.010,Y -239.736,Z 279.764,A 0.000,B 0.000,C 90.000,E1 317.595} C_DIS
LIN {X 0.016,Y -249.789,Z 279.746,A 0.000,B 0.000,C 90.000,E1 314.271} C_DIS
LIN {X -0.021,Y -260.871,Z 279.728,A 0.000,B 0.000,C 90.000,E1 311.024} C_DIS
LIN {X 0.123,Y -273.059,Z 279.710,A 0.000,B 0.000,C 90.000,E1 307.810} C_DIS
LIN {X -0.180,Y -285.104,Z 279.695,A 0.000,B 0.000,C 90.000,E1 305.105} C_DIS
LIN {X 0.133,Y -298.615,Z 279.680,A 0.000,B 0.000,C 90.000,E1 302.339} C_DIS
LIN {X -0.034,Y -315.465,Z 279.663,A 0.000,B 0.000,C 90.000,E1 299.411} C_DIS
LIN {X -0.041,Y -333.873,Z 279.647,A 0.000,B 0.000,C 90.000,E1 296.539} C_DIS
LIN {X 0.152,Y -346.640,Z 279.637,A 0.000,B 0.000,C 90.000,E1 294.643} C_DIS
LIN {X 0.187,Y -361.541,Z 279.625,A 0.000,B 0.000,C 90.000,E1 292.514} C_DIS
LIN {X -0.084,Y -376.682,Z 279.614,A 0.000,B 0.000,C 90.000,E1 290.482} C_DIS
LIN {X 0.201,Y -392.168,Z 279.602,A 0.000,B 0.000,C 90.000,E1 288.417} C_DIS
LIN {X 0.125,Y -405.509,Z 279.593,A 0.000,B 0.000,C 90.000,E1 286.732} C_DIS
LIN {X -0.107,Y -421.010,Z 279.582,A 0.000,B 0.000,C 90.000,E1 284.828} C_DIS
LIN {X -0.077,Y -427.563,Z 279.578,A 0.000,B 0.000,C 90.000,E1 284.008} C_DIS
LIN {X -0.126,Y -435.536,Z 279.572,A 0.000,B 0.000,C 90.000,E1 282.939} C_DIS
LIN {X 0.248,Y -442.783,Z 279.566,A 0.000,B 0.000,C 90.000,E1 281.827} C_DIS
LIN {X 0.195,Y -449.575,Z 279.560,A 0.000,B 0.000,C 90.000,E1 280.782} C_DIS
